(* IEC 61131-3 sources: MotionTestBenchMaster/Logical/00_AID/Libraries/Sidel_Libraries/Sidel, 28 files *)

(* ---- Types.typ ---- *)
TYPE
	AlarmCmd_Type : 	STRUCT
		ActionEn : BOOL := TRUE; (*If TRUE the action is performed; If FALSE the alarm is shown as a Message*)
		ByPassEn : BOOL;
		ByPass : BOOL;
		ActionDis : BOOL;
		Active : BOOL; (*If TRUE the alarm is activated.*)
		Visibility : BOOL := TRUE; (*If TRUE the HMI show the Alarm. The action will always performed*)
		DependentActive : BOOL; (*If TRUE the Alarm is deactivated by its master alarm V4.A.A.1.6.13*)
	END_STRUCT;
	AlarmCFG_Type : 	STRUCT
		Action : USINT;
		Category : USINT;
		OMAC_Code : UINT;
		OMAC_Index : UINT;
	END_STRUCT;
	ActionSum_Type : 	STRUCT
		Bit : UDINT;
	END_STRUCT;
	ActionSum_Enum :
		( (*V4.A.A.1.6.13*)
		ALR_NULL := 0, (*No Action, No Code*)
		ALR_MS_QuickStop := 1, (*Machine Stop: Fast deceleration ramp*)
		ALR_MS_NormalStop := 2, (*Machine Stop: Low deceleration ramp*)
		ALR_MS_QuickWithJog := 3, (*Machine Stop: Fast deceleration ramp + JOG Running Possible*)
		ALR_MS_NormalWithJog := 4, (*Machine Stop: Low deceleration ramp + JOG Running Possible*)
		ALR_MS_NormalWithJogMnt := 5, (*Machine Stop Auto Reset: Low deceleration ramp + JOG Running Possible*)
		ALR_CSR := 6, (*Container Stop Operator Reset: Immediate*)
		ALR_CSR_AfterSlowdown := 7, (*Container Stop Operator Reset: After Slowing*)
		ALR_CSR_StopAfterEmptying := 8, (*Container Stop Operator Reset: Emptying + Machine Normal Stop*)
		ALR_CSA := 9, (*Container Stop Auto Reset: Immediate*)
		ALR_CSA_AfterSlowdown := 10, (*Container Stop Auto Reset: After Slowing*)
		ALR_StartModeDisabled := 30, (*Start-Up Function Mode Disabled*)
		ALR_NoProduction := 31 (*No Action, Production Suspended (only Data Acquisition Code)*)
		);
	RCP_Management_Type : 	STRUCT
		Enable : BOOL; (*To HMI - Enable to download a recipe*)
		Started : BOOL; (*From HMI - Download Started*)
		Ended : BOOL; (*From HMI - Download Ended*)
		Received : BOOL; (*To HMI - Ended Received *)
		EditOnlineEnable : BOOL; (*To HMI - Edit Online Enabled*)
		EditOnlineActive : BOOL; (*From HMI - Edit Online Active*)
		ActiveRecipeName : STRING[70]; (*From HMI - Name of Actived Recipe*)
		RequestedRecipeName : STRING[70]; (*To HMI - Name of the requested recipe*)
		DownloadRequest : BOOL; (*To HMI - Request command to download a recipe*)
	END_STRUCT;
	RCP_Management_Step :
		(
		Wait_Download := 0,
		Download_Request := 1,
		Copy_To_Internal := 2,
		Download_Done := 3,
		Clear_Cmd := 4,
		Edit_Online := 10,
		Download_Error := 20
		);
	HMI_ITC_Page_Type : 	STRUCT
		PartnerID : USINT := 11;
		PageNum : USINT := 0;
	END_STRUCT;
	HMI_ITC_Data_Type : 	STRUCT
		PartnerID : USINT;
		ComType : USINT;
		ComAddress : STRING[35];
		ComSwap : BOOL;
		PageUp : HMI_ITC_PB_Type := (Visibility:=TRUE);
		PageDown : HMI_ITC_PB_Type := (Visibility:=TRUE);
		ComStatus : USINT;
		ComMask : HMI_ITC_SS2P_Type := (Visibility:=TRUE);
		DigitalIn : ARRAY[1..16]OF HMI_DigitalITC_Type;
		AnalogIn : ARRAY[1..4]OF HMI_AnalogITC_Type;
		DigitalOut : ARRAY[1..16]OF HMI_DigitalITC_Type;
		AnalogOut : ARRAY[1..4]OF HMI_AnalogITC_Type;
		ManActive : BOOL;
	END_STRUCT;
	HMI_AnalogITC_Type : 	STRUCT
		Visibility : BOOL;
		PV : REAL;
		Unit : STRING[10];
		Wait : BOOL;
		MinValue : REAL;
		MaxValue : REAL;
		Enable : BOOL;
		Man : BOOL;
		PV_Man : REAL;
		Description : STRING[100];
		Decimal : USINT;
	END_STRUCT;
	HMI_DigitalITC_Type : 	STRUCT
		Visibility : BOOL;
		Enable : BOOL;
		Auto : BOOL := TRUE;
		LampState : BOOL;
		Alarm : BOOL;
		Wait : BOOL;
		Man : BOOL;
		Description : STRING[100];
	END_STRUCT;
	HMI_ITC_PB_Type : 	STRUCT  (*Push button (ON-OFF;) 0=OFF - 1=ON*)
		Enable : BOOL; (*State: Command Enabled*)
		LampON : BOOL; (*State: Lamp Command ON*)
		Blink : BOOL; (*State: Blink LampOn*)
		Visibility : BOOL; (*Configuration: Present*)
		ON : BOOL; (*Command: Push Button ON*)
	END_STRUCT;
	HMI_ITC_SS2P_Type : 	STRUCT  (*Selector 2 position (Auto-Man; ON-OFF;) 0=Auto/OFF - 1=Man/ON*)
		Enable : BOOL; (*State: Command Enabled*)
		LampON : BOOL; (*State: Lamp Command ON*)
		Blink : BOOL; (*State: Blink LampOn*)
		Visibility : BOOL; (*Configuration: Present*)
		ON : BOOL; (*Command: Push Button ON*)
	END_STRUCT;
	IO_TimeClock_Type : 	STRUCT
		Seconds : UDINT;
		Nanoseconds : UDINT;
	END_STRUCT;
	Counters_Type : 	STRUCT
		CounterValue : UDINT;
		CounterTime : CounterTime_Type;
		StartDate : DINT;
	END_STRUCT;
	CounterTime_Type : 	STRUCT
		Day : UINT;
		Hour : USINT;
		Min : USINT;
		Sec : USINT;
	END_STRUCT;
	HMI_ComboBoxElements_Type : 	STRUCT
		Present : BOOL;
		Name : STRING[20];
	END_STRUCT;
	SEQ_StepConfig_Type : 	STRUCT
		T_TimePr : UINT;
		TO_TimePr : UINT;
		HMI_ID : UINT;
		TON_TimePr : UINT;
		Laps_Request : UINT;
		Cycle_Pr : UINT;
		TON_TimeSTART : BOOL;
		T_TimeSTART : BOOL;
		T_TimeSTOP : BOOL;
		T_TimeRESET : BOOL;
		Laps_Counter_Enable : BOOL;
		Cycle_RESET : BOOL;
	END_STRUCT;
	SIKO_MASTER_Type : 	STRUCT  (* *) (* *) (*13*)
		InPosition : BOOL; (*1 - The motor is in position*) (* *) (*14*)
		PositioningInProgress : BOOL; (*1 - The positioning task is in progress*) (* *) (*15*)
		CalibrationDone : BOOL; (*1 - The calibration operation is done*) (* *) (*16*)
		MotorDisabled : BOOL; (*1 - The motor is disabled*) (* *) (*17*)
		AbortPositioning : BOOL; (*1 - The current positioning is aborted*) (* *) (*18*)
		CalibrationInProgress : BOOL; (*1 - The calibration Process is in progress*) (* *) (*19*)
		Spare_06 : BOOL; (* *) (* *) (*20*)
		Spare_07 : BOOL; (* *) (* *) (*21*)
		JogForward : BOOL; (*1 - Jog Forward Command*) (* *) (*22*)
		JogBackward : BOOL; (*1 - Jog Backward Command*) (* *) (*23*)
		StartPositioning : BOOL; (*Positive Edge - Start positioning*) (* *) (*24*)
		StartRead : BOOL; (*Positive Edge - Start read parameter from the drive*) (* *) (*25*)
		StartWrite : BOOL; (*Positive Edge - Start write parameter from the drive*) (* *) (*26*)
		Calibrate : BOOL; (*Positive Edge - Calibrate command. (Calibrate value => Current pos)*) (* *) (*27*)
		Enable : BOOL; (*0 - Disable the motor; 1 - Enable motor*) (* *) (*28*)
		Spare_17 : BOOL; (* *) (* *) (*29*)
		ReadOrWriteError : BOOL; (*1 - A read or wirte error has occured*) (* *) (*30*)
		IllegalOperation : BOOL; (*1 - An illegal operation has occurred*) (* *) (*31*)
		DeviceOutsideSwLimit : BOOL; (*1 - The device is outside the sw limit*) (* *) (*32*)
		OnError : BOOL; (*1 - The motor is on error (current, temperature too high, ...)*) (* *) (*33*)
		TargetOutsideSwLimit : BOOL; (*1 - The target position is outside the sw limit (no movement is possible)*) (* *) (*34*)
		CommunicationFault : BOOL; (*1 - Comunication fault*) (* *) (*35*)
		Spare_26 : BOOL; (* *) (* *) (*36*)
		Warning : BOOL; (*1 - Warning present*) (* *) (*37*)
		EmergencyOkFbk : BOOL; (*Emergency ok feedback*) (* *) (*38*)
		WriteEnabled : BOOL; (*1 - Write process is enabled*) (* *) (*39*)
		ReadOrWriteInProgress : BOOL; (* *) (* *) (*40*)
		Spare_33 : BOOL; (* *) (* *) (*41*)
		Spare_34 : BOOL; (* *) (* *) (*42*)
		Spare_35 : BOOL; (* *) (* *) (*43*)
		Spare_36 : BOOL; (* *) (* *) (*44*)
		Spare_37 : BOOL; (* *) (* *) (*45*)
		TargetPos : REAL; (* *) (* *) (*46*)
		CurrentPos : REAL; (* *) (* *) (*47*)
		Data : SIKO_DATA_Type; (* *) (* *) (*48*)
	END_STRUCT;
	SIKO_DATA_Type : 	STRUCT  (* *) (* *) (*50*)
		OperationMode : INT; (*r/w - address:396hex - value: 2 - Don't change!!!!!!!!!!!!!!!!!!!!!!!!!!!!!!*) (* *) (*51*)
		PGain : INT; (*r/w - address:3e8hex*) (* *) (*52*)
		IGain : INT; (*r/w - address:3e9hex*) (* *) (*53*)
		DGain : INT; (*r/w - address:3eahex*) (* *) (*54*)
		VPos : INT; (*r/w - address:3echex*) (* *) (*55*)
		APos : INT; (*r/w - address:3ebhex*) (* *) (*56*)
		VJog : INT; (*r/w - address:3f0hex*) (* *) (*57*)
		SpareInt : INT; (* *) (* *) (*58*)
		GearIn : INT; (*r/w - address:3f2hex*) (* *) (*59*)
		GearOut : INT; (*r/w - address:3f3hex*) (* *) (*60*)
		SpindlePitch : INT; (*r/w - address:3f4hex*) (* *) (*61*)
		SenseOfRotation : INT; (*r/w - address:3f5hex*) (* *) (*62*)
		UpperLimit : REAL; (*r/w - address:3f8hex*) (* *) (*63*)
		LowerLimit : REAL; (*r/w - address:3f9hex*) (* *) (*64*)
		CalibrationValue : REAL; (*r/w - address:3fahex*) (* *) (*65*)
		SystemStatusWord : INT; (*r - address:3fchex*) (* *) (*66*)
		FaultBuffer0 : UINT; (*r - address:3b1 sub: 0*) (* *) (*67*)
		FaultBuffer1 : UINT; (*r - address:3b1 sub: 1*) (* *) (*68*)
		FaultBuffer2 : UINT; (*r - address:3b1 sub: 2*) (* *) (*69*)
		FaultBuffer3 : UINT; (*r - address:3b1 sub: 3*) (* *) (*70*)
		FaultBuffer4 : UINT; (*r - address:3b1 sub: 4*) (* *) (*71*)
		FaultBuffer5 : UINT; (*r - address:3b1 sub: 5*) (* *) (*72*)
		FaultBuffer6 : UINT; (*r - address:3b1 sub: 6*) (* *) (*73*)
		FaultBuffer7 : UINT; (*r - address:3b1 sub: 7*) (* *) (*74*)
		FaultBuffer8 : UINT; (*r - address:3b1 sub: 8*) (* *) (*75*)
		FaultBuffer9 : UINT; (*r - address:3b1 sub: 9*) (* *) (*76*)
		TimeoutPositioning : TIME; (* *) (* *) (*77*)
		PosWindows : REAL; (*r/w - address:3f1hex*) (* *) (*78*)
	END_STRUCT;
	SIKO_COM_Type : 	STRUCT  (* *) (* *) (*80*)
		FLR_SIKO : FLR_SIKO_Type; (* *) (* *) (*81*)
		SIKO_FLR : SIKO_FLR_Type; (* *) (* *) (*82*)
	END_STRUCT;
	FLR_SIKO_Type : 	STRUCT  (* *) (* *) (*84*)
		PKE : UINT; (* *) (* *) (*85*)
		IND : UINT; (* *) (* *) (*86*)
		PWE_H : UINT; (* *) (* *) (*87*)
		PWE_L : UINT; (* *) (* *) (*88*)
		STW : UINT; (* *) (* *) (*89*)
		HSW_H : UINT; (* *) (* *) (*90*)
		HSW_L : UINT; (* *) (* *) (*91*)
	END_STRUCT;
	SIKO_FLR_Type : 	STRUCT  (* *) (* *) (*93*)
		PKE : UINT; (* *) (* *) (*94*)
		IND : UINT; (* *) (* *) (*95*)
		PWE_H : UINT; (* *) (* *) (*96*)
		PWE_L : UINT; (* *) (* *) (*97*)
		ZSW : UINT; (* *) (* *) (*98*)
		HIW_H : UINT; (* *) (* *) (*99*)
		HIW_L : UINT; (* *) (* *) (*100*)
	END_STRUCT;
	AlarmAreaCfg_Type : 	STRUCT  (*V4.A.A.1.6.13*)
		From : UINT;
		To : UINT;
	END_STRUCT;
END_TYPE

(* ---- ComboBox.st ---- *)
FUNCTION ComboBoxString
	OUT_ComboString := '';
	FOR VAR_ElementsIndex := 0 TO 16 DO
		IF IN_ElementsStructure[VAR_ElementsIndex].Present THEN
			itoa(USINT_TO_DINT(VAR_ElementsIndex), ADR(VAR_StrIndex));
			VAR_StrComma 		:= ',';
			VAR_StrSemicolun 	:= ';';
			strcat(ADR(OUT_ComboString), ADR(VAR_StrIndex));
			strcat(ADR(OUT_ComboString), ADR(VAR_StrComma));
			strcat(ADR(OUT_ComboString), ADR(IN_ElementsStructure[VAR_ElementsIndex].Name));
			strcat(ADR(OUT_ComboString), ADR(VAR_StrSemicolun));
		END_IF
	END_FOR
	ComboBoxString := TRUE;
END_FUNCTION

(* ---- FC_Counter.st ---- *)
FUNCTION FC_Counter
	IF(IN_Clock1Hz) AND IN_TimeCondition THEN
		FC_Counter	:= TRUE;
		IN_OUT_CounterPartialStruct.CounterTime.Sec	:= IN_OUT_CounterPartialStruct.CounterTime.Sec + 1;
		IF (IN_OUT_CounterPartialStruct.CounterTime.Sec >= 60) THEN
			IN_OUT_CounterPartialStruct.CounterTime.Sec	:= 0;
			IN_OUT_CounterPartialStruct.CounterTime.Min	:= IN_OUT_CounterPartialStruct.CounterTime.Min + 1;
			IF IN_OUT_CounterPartialStruct.CounterTime.Min >= 60 THEN
				IN_OUT_CounterPartialStruct.CounterTime.Min	:= 0;
				IN_OUT_CounterPartialStruct.CounterTime.Hour	:= IN_OUT_CounterPartialStruct.CounterTime.Hour + 1;
				IF IN_OUT_CounterPartialStruct.CounterTime.Hour >= 24 THEN
					IN_OUT_CounterPartialStruct.CounterTime.Hour	:= 0;
					IN_OUT_CounterPartialStruct.CounterTime.Day	:= IN_OUT_CounterPartialStruct.CounterTime.Day + 1;
				END_IF
			END_IF
		END_IF

		IN_OUT_CounterTotalStruct.CounterTime.Sec	:= IN_OUT_CounterTotalStruct.CounterTime.Sec + 1;
		IF (IN_OUT_CounterTotalStruct.CounterTime.Sec >= 60) THEN
			IN_OUT_CounterTotalStruct.CounterTime.Sec	:= 0;
			IN_OUT_CounterTotalStruct.CounterTime.Min	:= IN_OUT_CounterTotalStruct.CounterTime.Min + 1;
			IF IN_OUT_CounterTotalStruct.CounterTime.Min >= 60 THEN
				IN_OUT_CounterTotalStruct.CounterTime.Min	:= 0;
				IN_OUT_CounterTotalStruct.CounterTime.Hour	:= IN_OUT_CounterTotalStruct.CounterTime.Hour + 1;
				IF IN_OUT_CounterTotalStruct.CounterTime.Hour >= 24 THEN
					IN_OUT_CounterTotalStruct.CounterTime.Hour	:= 0;
					IN_OUT_CounterTotalStruct.CounterTime.Day	:= IN_OUT_CounterTotalStruct.CounterTime.Day + 1;
				END_IF
			END_IF
		END_IF
	END_IF

	IF IN_IncrementCondition THEN
		FC_Counter	:= TRUE;
		IN_OUT_CounterPartialStruct.CounterValue	:= IN_OUT_CounterPartialStruct.CounterValue + 1;
		IN_OUT_CounterTotalStruct.CounterValue		:= IN_OUT_CounterTotalStruct.CounterValue + 1;
	END_IF

	IF IN_Reset THEN
		FC_Counter	:= TRUE;
		IN_OUT_CounterPartialStruct.CounterTime.Sec		:= 0;
		IN_OUT_CounterPartialStruct.CounterTime.Min		:= 0;
		IN_OUT_CounterPartialStruct.CounterTime.Hour	:= 0;
		IN_OUT_CounterPartialStruct.CounterTime.Day		:= 0;
		IN_OUT_CounterPartialStruct.CounterValue		:= 0;
		IN_OUT_CounterPartialStruct.StartDate			:= DT_TO_DINT(IN_Date);
	ELSIF IN_OUT_CounterPartialStruct.StartDate = 0 THEN
		IN_OUT_CounterPartialStruct.StartDate		:= DT_TO_DINT(IN_Date);
	ELSIF IN_OUT_CounterTotalStruct.StartDate	= 0 THEN
		IN_OUT_CounterTotalStruct.StartDate		:= DT_TO_DINT(IN_Date);
	END_IF
END_FUNCTION

(* ---- FC_Parity.st ---- *)
FUNCTION FC_Parity
	FC_Parity := NOT IN_Value.0;
END_FUNCTION

(* ---- FC_Reminder.st ---- *)
(* Reminder With Minimum Value *)
FUNCTION FC_ReminderShift
	LocalDivisor	:= SEL(Divisor<>0, 1, Divisor);

	ReminderA	:= (Dividend - ((Dividend / LocalDivisor) * LocalDivisor));
	ReminderB	:= (ReminderA + Divisor - ((ReminderA + LocalDivisor) / LocalDivisor) * LocalDivisor);
	ReminderC	:= (ReminderB + Start - ((ReminderB + Start) / LocalDivisor) * LocalDivisor);

	FC_ReminderShift	:= SEL(ReminderC <> 0, LocalDivisor, ReminderC);
END_FUNCTION

(* ---- FC_SpeedCheck.st ---- *)
FUNCTION FC_SpeedCheck
	CASE IN_Mode OF
		CST_EQ:	(* Actual speed equal to requested *)
			FC_SpeedCheck := (IN_SpeedAct >= (IN_SpeedReq * 0.9)) AND (IN_SpeedAct <= (IN_SpeedReq / 0.9));

		CST_GE:	(* Actual speed greater then requested *)
			FC_SpeedCheck := IN_SpeedAct >= IN_SpeedReq * 0.9;

		CST_LE:	(* Actual speed lower then requested *)
			FC_SpeedCheck := IN_SpeedAct <= IN_SpeedReq / 0.9;

		CST_GT:	(* Actual speed greater then requested *)
			FC_SpeedCheck := IN_SpeedAct > IN_SpeedReq * 0.9;

		CST_LT:	(* Actual speed lower then requested *)
			FC_SpeedCheck := IN_SpeedAct < IN_SpeedReq / 0.9;

		ELSE
			FC_SpeedCheck := FALSE;
	END_CASE
END_FUNCTION

(* ---- FC_Timer.st ---- *)
FUNCTION FC_IncTimer
	IF IN_Reset THEN
		FC_IncTimer	:= TRUE;
		IN_OUT_CounterStruct.Sec	:= 0;
		IN_OUT_CounterStruct.Min	:= 0;
		IN_OUT_CounterStruct.Hour	:= 0;
		IN_OUT_CounterStruct.Day	:= 0;
	ELSIF(IN_Clock1Hz) AND IN_Condition THEN
		FC_IncTimer	:=	TRUE;
		IN_OUT_CounterStruct.Sec	:= IN_OUT_CounterStruct.Sec + 1;
		IF (IN_OUT_CounterStruct.Sec >= 60) THEN
			IN_OUT_CounterStruct.Sec	:= 0;
			IN_OUT_CounterStruct.Min	:= IN_OUT_CounterStruct.Min + 1;
			IF IN_OUT_CounterStruct.Min >= 60 THEN
				IN_OUT_CounterStruct.Min	:= 0;
				IN_OUT_CounterStruct.Hour	:= IN_OUT_CounterStruct.Hour + 1;
				IF IN_OUT_CounterStruct.Hour >= 24 THEN
					IN_OUT_CounterStruct.Hour	:= 0;
					IN_OUT_CounterStruct.Day	:= IN_OUT_CounterStruct.Day + 1;
				END_IF
			END_IF
		END_IF
	ELSE
		FC_IncTimer	:= FALSE;
	END_IF
END_FUNCTION

FUNCTION FC_MacaoTimer
	IF IN_Reset THEN
		IN_OUT_Counter	:= 0;
	ELSIF IN_Clock1Hz AND IN_Condition THEN
		IN_OUT_Counter	:= IN_OUT_Counter + 1;
	END_IF
	FC_MacaoTimer := TRUE;
END_FUNCTION

(* ---- LftConAirPress.st ---- *)
FUNCTION LftConAirPressSp
	VAR_PistonSurface 	:= amPI * (EXPT(CST_PistonDiameterExt, 2) - EXPT(CST_PistonDiameterInt, 2)) / 4.0;
	VAR_DeltaPProduct 	:= (EXPT(57.0, 2) - EXPT(RcpCanDiameter, 2)) * amPI / 4.0 * RcpPressureSp / 10.0;
	VAR_DeltaPrexPist  	:= (ABS(VAR_DeltaPProduct * 1000000.0 / VAR_PistonSurface / 100000.0)) * BOOL_TO_REAL((RcpCanDiameter > 57.0));
	VAR_PbasePiston 	:= CST_PistonSpringStrengthRse / (VAR_PistonSurface / 100.0) / 10;
	LftConAirPressSp	:= VAR_PbasePiston + VAR_DeltaPrexPist + 1.5;
END_FUNCTION

(* ---- AlarmScheduler.st ---- *)
FUNCTION_BLOCK AlarmScheduler
	//V4.A.A.1.6.13
	memset(ADR(AlarmActionTemp), 0, SIZEOF(AlarmActionTemp));

	FOR x := 0 TO 24 DO//V1.7.2
		IF AlarmAreaCfg[x].From = 0 OR AlarmAreaCfg[x].To = 0 THEN
		ELSE
			FOR i := MAX(0, AlarmAreaCfg[x].From - 1) TO MAX(AlarmAreaCfg[x].To - 1, AlarmAreaCfg[x].From - 1) DO

				Alarm ACCESS AdrAlarm + (SIZEOF(Alarm) * i);
				AlarmCFG ACCESS AdrAlarmCFG + (SIZEOF(AlarmCFG) * i);
				AlarmOldStatus ACCESS AdrAlarmOldStatus + (SIZEOF(AlarmOldStatus) * i);
				HMI ACCESS AdrHMI + (SIZEOF(HMI) * i);

				IF FirstAlarmActive.OMAC_Index = AlarmCFG.OMAC_Index THEN
					memset(ADR(FirstAlarmActive), 0, SIZEOF(FirstAlarmActive));
				END_IF

				IF FirstExternalAlarmActive.OMAC_Index = AlarmCFG.OMAC_Index THEN
					memset(ADR(FirstExternalAlarmActive), 0, SIZEOF(FirstExternalAlarmActive));
				END_IF

				IF FirstAlarmActive.OMAC_Index = 0      AND Alarm.Active AND
					(Alarm.ActionEn AND NOT Alarm.ByPass) AND
					(AlarmCFG.Action <> 0) AND (AlarmCFG.Action <> 67) AND
					NOT Alarm.DependentActive THEN
					FirstAlarmActive := AlarmCFG;
				END_IF

				IF FirstExternalAlarmActive.OMAC_Index = 0      AND Alarm.Active AND
					(Alarm.ActionEn AND NOT Alarm.ByPass) AND
					(AlarmCFG.Action <> 0) AND (AlarmCFG.Category = 3) AND
					NOT Alarm.DependentActive THEN
					FirstExternalAlarmActive := AlarmCFG;
				END_IF

				IF Alarm.Active AND (Alarm.ActionEn AND NOT Alarm.ByPass AND Alarm.Visibility) AND
					NOT AlarmOldStatus AND NOT CriticalAcknoledgeRequest AND
					(AlarmCFG.Action > 0 AND AlarmCFG.Action < 32)	AND
					NOT Alarm.DependentActive THEN
					CriticalAcknoledgeRequest := AlarmCFG.Action <> 6; //ALARM SCHEDULER V4_03:ESCLUSIONE DEGLI ALLARMI DI SBLOCCO PORTE
				END_IF

				IF Alarm.Active AND (Alarm.ActionEn AND NOT Alarm.ByPass AND Alarm.Visibility) AND
					NOT AlarmOldStatus AND NOT AlarmAcknoledgeRequest AND
					(AlarmCFG.Action >= 32 AND AlarmCFG.Action < 64)	AND
					NOT Alarm.DependentActive THEN
					AlarmAcknoledgeRequest := TRUE;
				END_IF

				Alarm.ActionDis := NOT Alarm.ActionEn;

				HMI.0			:= Alarm.ActionEn;
				HMI.1			:= Alarm.ByPassEn;
				HMI.2;
				HMI.3;
				Alarm.ByPass	:= HMI.4;
				HMI.5			:= Alarm.ActionDis;
				HMI.6			:= Alarm.Active;
				HMI.7			:= Alarm.Visibility;

				CASE AlarmCFG.Action OF

					0:
						AlarmActionTemp.Bit.ALR_NULL					:= Alarm.Active AND NOT Alarm.DependentActive OR AlarmActionTemp.Bit.ALR_NULL;
					1:
						AlarmActionTemp.Bit.ALR_MS_QuickStop			:= Alarm.Active AND (Alarm.ActionEn AND NOT Alarm.ByPass AND NOT Alarm.DependentActive) OR AlarmActionTemp.Bit.ALR_MS_QuickStop;
					2:
						AlarmActionTemp.Bit.ALR_MS_NormalStop			:= Alarm.Active AND (Alarm.ActionEn AND NOT Alarm.ByPass AND NOT Alarm.DependentActive) OR AlarmActionTemp.Bit.ALR_MS_NormalStop;
					3:
						AlarmActionTemp.Bit.ALR_MS_QuickWithJog			:= Alarm.Active AND (Alarm.ActionEn AND NOT Alarm.ByPass AND NOT Alarm.DependentActive) OR AlarmActionTemp.Bit.ALR_MS_QuickWithJog;
					4:
						AlarmActionTemp.Bit.ALR_MS_NormalWithJog		:= Alarm.Active AND (Alarm.ActionEn AND NOT Alarm.ByPass AND NOT Alarm.DependentActive) OR AlarmActionTemp.Bit.ALR_MS_NormalWithJog;
					6:
						AlarmActionTemp.Bit.ALR_MS_NormalWithJogMnt		:= Alarm.Active AND (Alarm.ActionEn AND NOT Alarm.ByPass AND NOT Alarm.DependentActive) OR AlarmActionTemp.Bit.ALR_MS_NormalWithJogMnt;
					10:
						AlarmActionTemp.Bit.ALR_CSR_StopAfterEmptying	:= Alarm.Active AND (Alarm.ActionEn AND NOT Alarm.ByPass AND NOT Alarm.DependentActive) OR AlarmActionTemp.Bit.ALR_CSR_StopAfterEmptying;
					32:
						AlarmActionTemp.Bit.ALR_CSR						:= Alarm.Active AND (Alarm.ActionEn AND NOT Alarm.ByPass AND NOT Alarm.DependentActive) OR AlarmActionTemp.Bit.ALR_CSR;
					33:
						AlarmActionTemp.Bit.ALR_CSR_AfterSlowdown		:= Alarm.Active AND (Alarm.ActionEn AND NOT Alarm.ByPass AND NOT Alarm.DependentActive) OR AlarmActionTemp.Bit.ALR_CSR_AfterSlowdown;
					64:
						AlarmActionTemp.Bit.ALR_CSA						:= Alarm.Active AND (Alarm.ActionEn AND NOT Alarm.ByPass AND NOT Alarm.DependentActive) OR AlarmActionTemp.Bit.ALR_CSA;
					65:
						AlarmActionTemp.Bit.ALR_CSA_AfterSlowdown		:= Alarm.Active AND (Alarm.ActionEn AND NOT Alarm.ByPass AND NOT Alarm.DependentActive) OR AlarmActionTemp.Bit.ALR_CSA_AfterSlowdown;
					81:
						AlarmActionTemp.Bit.ALR_StartModeDisabled		:= Alarm.Active AND (Alarm.ActionEn AND NOT Alarm.ByPass AND NOT Alarm.DependentActive) OR AlarmActionTemp.Bit.ALR_StartModeDisabled;
					86:
						AlarmActionTemp.Bit.ALR_NoProduction			:= Alarm.Active AND (Alarm.ActionEn AND NOT Alarm.ByPass AND NOT Alarm.DependentActive) OR AlarmActionTemp.Bit.ALR_NoProduction;

					ELSE
						AlarmActionTemp.Bit.ALR_NULL					:= Alarm.Active AND NOT Alarm.DependentActive OR AlarmActionTemp.Bit.ALR_NULL;
				END_CASE

				//EXTRACTION OF FIRST ALARM FOR EACH CATEGORY
				IF FirstCriticalAlarmActive.OMAC_Index = AlarmCFG.OMAC_Index THEN//V4.A.A.1.7.0
					memset(ADR(FirstCriticalAlarmActive), 0, SIZEOF(FirstCriticalAlarmActive));
				END_IF

				IF FirstAlertAlarmActive.OMAC_Index = AlarmCFG.OMAC_Index THEN//V4.A.A.1.7.0
					memset(ADR(FirstAlertAlarmActive), 0, SIZEOF(FirstAlertAlarmActive));
				END_IF

				IF FirstExtCriticalAlarmActive.OMAC_Index = AlarmCFG.OMAC_Index THEN//V4.A.A.1.7.0
					memset(ADR(FirstExtCriticalAlarmActive), 0, SIZEOF(FirstExtCriticalAlarmActive));
				END_IF

				IF FirstExtAlertAlarmActive.OMAC_Index = AlarmCFG.OMAC_Index THEN//V4.A.A.1.7.0
					memset(ADR(FirstExtAlertAlarmActive), 0, SIZEOF(FirstExtAlertAlarmActive));
				END_IF
				IF FirstCsAlarmActive.OMAC_Index = AlarmCFG.OMAC_Index THEN//V4.A.A.1.7.0
					memset(ADR(FirstCsAlarmActive), 0, SIZEOF(FirstCsAlarmActive));
				END_IF
				//V4.A.A.1.7.0
				IF FirstCriticalAlarmActive.OMAC_Index = 0	AND Alarm.Active		AND
					(Alarm.ActionEn					AND NOT Alarm.ByPass)		AND
					(AlarmCFG.Action > 0)			AND (AlarmCFG.Action <= 31)	AND (AlarmCFG.Category <> 3) AND
					NOT Alarm.DependentActive THEN
					FirstCriticalAlarmActive := AlarmCFG;
				END_IF
				//V4.A.A.1.7.0
				IF FirstAlertAlarmActive.OMAC_Index = 0	AND Alarm.Active			AND
					(Alarm.ActionEn					AND NOT Alarm.ByPass)		AND
					(AlarmCFG.Action >= 32)			AND (AlarmCFG.Action <= 63)	AND (AlarmCFG.Category <> 3) AND
					NOT Alarm.DependentActive THEN
					FirstAlertAlarmActive := AlarmCFG;
				END_IF
				//V4.A.A.1.7.0
				IF FirstExtCriticalAlarmActive.OMAC_Index = 0	AND Alarm.Active			AND
					(Alarm.ActionEn							AND NOT Alarm.ByPass)		AND
					(AlarmCFG.Action > 0)			AND (AlarmCFG.Action <= 31)	AND (AlarmCFG.Category = 3)	AND
					NOT Alarm.DependentActive THEN
					FirstExtCriticalAlarmActive := AlarmCFG;
				END_IF
				//V4.A.A.1.7.0
				IF FirstExtAlertAlarmActive.OMAC_Index = 0	AND Alarm.Active			AND
					(Alarm.ActionEn							AND NOT Alarm.ByPass)		AND
					(AlarmCFG.Action >= 32)			AND (AlarmCFG.Action <= 63)	AND (AlarmCFG.Category = 3)	AND
					NOT Alarm.DependentActive THEN
					FirstExtAlertAlarmActive := AlarmCFG;
				END_IF
				//V4.A.A.1.7.0
				IF FirstCsAlarmActive.OMAC_Index = 0	AND Alarm.Active			AND
					(Alarm.ActionEn							AND NOT Alarm.ByPass)		AND
					(AlarmCFG.Action >= 64)			AND (AlarmCFG.Action <= 65)	AND
					NOT Alarm.DependentActive THEN
					FirstCsAlarmActive := AlarmCFG;
				END_IF
				//END EXTRACTION

				AlarmOldStatus := Alarm.Active AND (Alarm.ActionEn AND NOT Alarm.ByPass AND NOT Alarm.DependentActive);
			END_FOR
		END_IF
	END_FOR

	AlarmAction	:= AlarmActionTemp;
END_FUNCTION_BLOCK

FUNCTION_BLOCK FirstAlarmCombiner
	IF (FirstAlarmActive.OMAC_Index >= SkidAlarmFrom) AND (FirstAlarmActive.OMAC_Index <= SkidAlarmTo) THEN
		memset(ADR(FirstAlarmActive), 0, SIZEOF(FirstAlarmActive));
	END_IF

	IF (FirstExternalAlarmActive.OMAC_Index >= SkidAlarmFrom) AND (FirstExternalAlarmActive.OMAC_Index <= SkidAlarmTo) THEN
		memset(ADR(FirstExternalAlarmActive), 0, SIZEOF(FirstExternalAlarmActive));
	END_IF

	IF SkidFirstAlarm <> 0 AND FirstAlarmActive.OMAC_Index = 0 THEN
		FirstAlarmActive.OMAC_Index := SkidFirstAlarm;
	END_IF

	IF SkidFirstExternalAlarm <> 0 AND FirstExternalAlarmActive.OMAC_Index = 0 THEN
		FirstExternalAlarmActive.OMAC_Index := SkidFirstExternalAlarm;
	END_IF
END_FUNCTION_BLOCK

(* ---- AnalogTotalizer.st ---- *)
FUNCTION_BLOCK AnalogTotalizer
	RTInfo(enable := TRUE);

	CASE IN_ConfigType OF
		0:
			VAR_AuxPulse := IN_PulseWeight * BOOL_TO_REAL(EDGEPOS(IN_Pulse));
		1:
			VAR_AuxPulse := IN_AnalogPV * UDINT_TO_REAL(RTInfo.cycle_time) /1000000;
		2:
			VAR_AuxPulse := IN_AnalogPV * UDINT_TO_REAL(RTInfo.cycle_time) /1000000 / 60;
		3:
			VAR_AuxPulse := IN_AnalogPV * UDINT_TO_REAL(RTInfo.cycle_time) /1000000 / 3600;
	END_CASE

	OUT_TotalCounter := VAR_AuxPulse + OUT_TotalCounter;

	IF IN_Reset THEN
		OUT_TotalCounter := 0.0;
	END_IF
END_FUNCTION_BLOCK

(* ---- Blink.st ---- *)
FUNCTION_BLOCK FB_Blinker
	VAR_TimeValue	:= REAL_TO_TIME((1.0 / IN_Freq) * 1000);

	TMR_TON_OnDelay(IN:= NOT OUT,	PT:= VAR_TimeValue / 2);
	TMR_TON_OffDelay(IN:= OUT,		PT:= VAR_TimeValue / 2);

	IF TMR_TON_OnDelay.Q THEN
		OUT	:= TRUE;
	ELSIF TMR_TON_OffDelay.Q THEN
		OUT	:= FALSE;
	END_IF
END_FUNCTION_BLOCK

(* ---- CyclicActivation.st ---- *)
FUNCTION_BLOCK CyclicActivation
	VAR_RtInfo(enable:=TRUE);
	VAR_CycleCounter	:= MAX(1, VAR_CycleCounter + 1);
	OUT_A	:= FALSE;
	OUT_B	:= FALSE;

	TMR_TON_CycleA(	IN := VAR_Cycle,
	PT := (IN_CycleTime / 2) - UDINT_TO_TIME(VAR_RtInfo.cycle_time / 1000));

	TMR_TON_CycleB(	IN := NOT VAR_Cycle,
	PT := (IN_CycleTime / 2) - UDINT_TO_TIME(VAR_RtInfo.cycle_time / 1000));

	IF TMR_TON_CycleA.Q THEN
		OUT_A		:= TRUE;
		VAR_Cycle	:= FALSE;
	ELSIF TMR_TON_CycleB.Q THEN
		OUT_B		:= TRUE;
		VAR_Cycle	:= TRUE;
	ELSE
		RETURN;
	END_IF

	VAR_CycleTime	:= (UDINT_TO_REAL(VAR_RtInfo.cycle_time) * VAR_CycleCounter) / 1000000.0;
	VAR_CycleCounter 	:= 0.0;
	memset(ADR(TMR_TON_CycleA), 0, SIZEOF(TMR_TON_CycleA));
	memset(ADR(TMR_TON_CycleB), 0, SIZEOF(TMR_TON_CycleB));
END_FUNCTION_BLOCK

(* ---- FB_Counter.st ---- *)
FUNCTION_BLOCK FB_Counter
	IF(IN_Clock1Hz) AND IN_TimeCondition THEN
		IN_OUT_CounterPartialStruct.CounterTime.Sec	:= IN_OUT_CounterPartialStruct.CounterTime.Sec + 1;
		IF (IN_OUT_CounterPartialStruct.CounterTime.Sec >= 60) THEN
			IN_OUT_CounterPartialStruct.CounterTime.Sec	:= 0;
			IN_OUT_CounterPartialStruct.CounterTime.Min	:= IN_OUT_CounterPartialStruct.CounterTime.Min + 1;
			IF IN_OUT_CounterPartialStruct.CounterTime.Min >= 60 THEN
				IN_OUT_CounterPartialStruct.CounterTime.Min	:= 0;
				IN_OUT_CounterPartialStruct.CounterTime.Hour	:= IN_OUT_CounterPartialStruct.CounterTime.Hour + 1;
				IF IN_OUT_CounterPartialStruct.CounterTime.Hour >= 24 THEN
					IN_OUT_CounterPartialStruct.CounterTime.Hour	:= 0;
					IN_OUT_CounterPartialStruct.CounterTime.Day	:= IN_OUT_CounterPartialStruct.CounterTime.Day + 1;
				END_IF
			END_IF
		END_IF

		IN_OUT_CounterTotalStruct.CounterTime.Sec	:= IN_OUT_CounterTotalStruct.CounterTime.Sec + 1;
		IF (IN_OUT_CounterTotalStruct.CounterTime.Sec >= 60) THEN
			IN_OUT_CounterTotalStruct.CounterTime.Sec	:= 0;
			IN_OUT_CounterTotalStruct.CounterTime.Min	:= IN_OUT_CounterTotalStruct.CounterTime.Min + 1;
			IF IN_OUT_CounterTotalStruct.CounterTime.Min >= 60 THEN
				IN_OUT_CounterTotalStruct.CounterTime.Min	:= 0;
				IN_OUT_CounterTotalStruct.CounterTime.Hour	:= IN_OUT_CounterTotalStruct.CounterTime.Hour + 1;
				IF IN_OUT_CounterTotalStruct.CounterTime.Hour >= 24 THEN
					IN_OUT_CounterTotalStruct.CounterTime.Hour	:= 0;
					IN_OUT_CounterTotalStruct.CounterTime.Day	:= IN_OUT_CounterTotalStruct.CounterTime.Day + 1;
				END_IF
			END_IF
		END_IF
	END_IF

	IF IN_IncrementCondition THEN
		tempReal := tempReal + IN_PulseWeight;
		IF tempReal >= 1.0 THEN
			IN_OUT_CounterPartialStruct.CounterValue	:= IN_OUT_CounterPartialStruct.CounterValue + TRUNC(tempReal);
			IN_OUT_CounterTotalStruct.CounterValue		:= IN_OUT_CounterTotalStruct.CounterValue 	+ TRUNC(tempReal);
			tempReal := tempReal - (TRUNC(tempReal));
		END_IF
	END_IF

	IF IN_Reset THEN
		IN_OUT_CounterPartialStruct.CounterTime.Sec		:= 0;
		IN_OUT_CounterPartialStruct.CounterTime.Min		:= 0;
		IN_OUT_CounterPartialStruct.CounterTime.Hour	:= 0;
		IN_OUT_CounterPartialStruct.CounterTime.Day		:= 0;
		IN_OUT_CounterPartialStruct.CounterValue		:= 0;
		IN_OUT_CounterPartialStruct.StartDate			:= DT_TO_DINT(IN_Date);
	ELSIF IN_OUT_CounterPartialStruct.StartDate = 0 THEN
		IN_OUT_CounterPartialStruct.StartDate		:= DT_TO_DINT(IN_Date);
	ELSIF IN_OUT_CounterTotalStruct.StartDate	= 0 THEN
		IN_OUT_CounterTotalStruct.StartDate		:= DT_TO_DINT(IN_Date);
	END_IF
END_FUNCTION_BLOCK

(* ---- FB_Flip.st ---- *)
FUNCTION_BLOCK FB_Flip
	TON_Blink.IN := NOT TON_Blink.Q;
	TON_Blink.PT := t#1s;
	TON_Blink();

	IF EDGEPOS(TON_Blink.Q) THEN
		VAR_CyleOn 		:= FALSE;
		VAR_CyleCntOn	:= FALSE;
		VAR_CyleCntOff	:= FALSE;
		VAR_CyleOnTimeReset := FALSE;
		VAR_CyleOffTimeReset:= FALSE;
		VAR_CyleNrReset	:= FALSE;
		VAR_CycleNrDone	:= FALSE;
		CASE Command_State OF
			0:
				IF IN_CycleOn AND NOT IN_CyclePause THEN
					IF IN_CycleStartOffCount THEN
						Command_State := 2;
					ELSIF IN_CycleTimeOn > 0 THEN
						Command_State := 1;
					END_IF
				END_IF

			1:	//ON TIME
				VAR_CyleOn 		:= TRUE;
				VAR_CyleCntOn	:= TRUE;
				VAR_CyleOffTimeReset	:= TRUE;

				IF NOT IN_CycleOn THEN
					Command_State := 99; // //RESET CNT
				ELSIF IN_CyclePause THEN
					Command_State := 10; // PAUSE CMD
				ELSE
					IF VAR_CycleOnDone THEN
						VAR_CyleOnTimeReset := TRUE;
						IF IN_CycleLoop THEN
							IF IN_CycleTimeOff > 0 THEN
								Command_State := 2; //PAUSE TIME
							END_IF
						ELSE
							VAR_CycleNr 	:= MIN(VAR_CycleNr  +1, IN_CycleNr);
							 IF (IN_CycleNr = VAR_CycleNr) AND NOT IN_CycleLoop THEN
								Command_State := 3; // DONE
							ELSE
								Command_State := 2; //PAUSE TIME
							END_IF
						END_IF
					END_IF
				END_IF

			2: //PAUSE TIME

				VAR_CyleCntOff	:= NOT IN_CyclePause;
				VAR_CyleOnTimeReset	:= TRUE;

				IF NOT IN_CycleOn THEN
					Command_State := 99; // //RESET CNT
				ELSIF VAR_CycleOffDone AND NOT IN_CyclePause THEN
					VAR_CyleOffTimeReset := TRUE;
					IF VAR_CycleNrDone THEN
						Command_State := 3; // DONE
					ELSIF IN_CycleTimeOn > 0 THEN
						Command_State := 1; // ON TIME
					END_IF
				END_IF

			3: // DONE
				VAR_CycleNrDone	:= TRUE;
				IF NOT IN_CycleOn OR IN_CycleLoop THEN
					Command_State := 99; // //RESET CNT
				END_IF

			10: // PAUSE

				IF NOT IN_CycleOn THEN
					Command_State := 99; // //RESET CNT
				ELSIF NOT IN_CyclePause THEN
					Command_State := 1; // OFF
				END_IF

			99: //RESET CNT
				VAR_CyleOnTimeReset := TRUE;
				VAR_CyleOffTimeReset:= TRUE;
				VAR_CycleNr := 0;
				Command_State := 0; // OFF
		END_CASE

		IF VAR_CyleCntOn THEN
			VAR_CycleTimeOn := MIN(VAR_CycleTimeOn  +1, IN_CycleTimeOn);
			VAR_CycleOnDone := IN_CycleTimeOn = VAR_CycleTimeOn;
		ELSE
			VAR_CycleOnDone := FALSE;
		END_IF

		IF VAR_CyleCntOff THEN
			VAR_CycleTimeOff := MIN(VAR_CycleTimeOff +1, IN_CycleTimeOff);
			VAR_CycleOffDone := IN_CycleTimeOff = VAR_CycleTimeOff;
		ELSE
			VAR_CycleOffDone := FALSE;
		END_IF

		IF VAR_CyleOffTimeReset THEN
			VAR_CycleTimeOff := 0;
		END_IF
		IF VAR_CyleOnTimeReset THEN
			VAR_CycleTimeOn := 0;
		END_IF
		IF IN_CycleNrReset THEN
			VAR_CycleNr 	:= 0;
		END_IF

		Out 			:= VAR_CyleOn;
		OUT_CycleNr		:= VAR_CycleNr;
		OUT_CycleTimeOn	:= VAR_CycleTimeOn;
		OUT_CycleTimeOff:= VAR_CycleTimeOff;
		OUT_CycleDone 	:= VAR_CycleNrDone;
	END_IF
END_FUNCTION_BLOCK

(* ---- FB_ITC.st ---- *)
FUNCTION_BLOCK FB_HMI_ITC_DigitalBool
	VAR_ProgressiveId := INT_TO_UINT(FC_ReminderShift(UINT_TO_INT(Index), 16, 0));

	IF IN_ReadOnly OR IN_HMIAutoForce THEN
		VAR_Auto	:= TRUE;
		VAR_Man		:= FALSE;
	END_IF

	IF IN_IOType THEN
		ITC_IO 	:= SEL(VAR_Auto, VAR_Man, ITC);
	ELSE
		ITC 	:= SEL(VAR_Auto, VAR_Man, ITC_IO);
	END_IF

	IF VAR_OldPage <> HMI_Page.PageNum THEN
		VAR_PageSwitch	:= TRUE;
	END_IF

	IF (Index = (VAR_ProgressiveId + 16 * HMI_Page.PageNum)) AND IN_Visibility THEN
		IF VAR_PageSwitch THEN
			IF IN_IOType THEN
				HMI_Data.DigitalOut[VAR_ProgressiveId].Auto	:= VAR_Auto;
				HMI_Data.DigitalOut[VAR_ProgressiveId].Man	:= VAR_Man;
			ELSE
				HMI_Data.DigitalIn[VAR_ProgressiveId].Auto	:= VAR_Auto;
				HMI_Data.DigitalIn[VAR_ProgressiveId].Man	:= VAR_Man;
			END_IF
			VAR_PageSwitch	:= FALSE;
		END_IF

		IF IN_IOType THEN
			HMI_Data.DigitalOut[VAR_ProgressiveId].Visibility	:= IN_Visibility;
			HMI_Data.DigitalOut[VAR_ProgressiveId].Enable		:= NOT IN_ReadOnly AND NOT IN_HMIAutoForce;
			HMI_Data.DigitalOut[VAR_ProgressiveId].LampState	:= ITC_IO;
			HMI_Data.DigitalOut[VAR_ProgressiveId].Wait			:= IN_Wait;
			HMI_Data.DigitalOut[VAR_ProgressiveId].Alarm		:= IN_Alarm;
			HMI_Data.DigitalOut[VAR_ProgressiveId].Description	:= IN_Description;

			IF EDGEPOS(HMI_Data.DigitalOut[VAR_ProgressiveId].Auto) THEN
				HMI_Data.DigitalOut[VAR_ProgressiveId].Man := FALSE;
			ELSIF EDGEPOS(HMI_Data.DigitalOut[VAR_ProgressiveId].Man) THEN
				HMI_Data.DigitalOut[VAR_ProgressiveId].Auto := FALSE;
			END_IF

			IF IN_ReadOnly OR IN_HMIAutoForce THEN
				HMI_Data.DigitalOut[VAR_ProgressiveId].Auto	:= TRUE;
				HMI_Data.DigitalOut[VAR_ProgressiveId].Man	:= FALSE;
			END_IF

			VAR_Auto	:= HMI_Data.DigitalOut[VAR_ProgressiveId].Auto;
			VAR_Man		:= HMI_Data.DigitalOut[VAR_ProgressiveId].Man;
		ELSE
			HMI_Data.DigitalIn[VAR_ProgressiveId].Visibility	:= IN_Visibility;
			HMI_Data.DigitalIn[VAR_ProgressiveId].Enable		:= NOT IN_ReadOnly AND NOT IN_HMIAutoForce;
			HMI_Data.DigitalIn[VAR_ProgressiveId].LampState 	:= ITC;
			HMI_Data.DigitalIn[VAR_ProgressiveId].Wait			:= IN_Wait;
			HMI_Data.DigitalIn[VAR_ProgressiveId].Alarm			:= IN_Alarm;
			HMI_Data.DigitalIn[VAR_ProgressiveId].Description	:= IN_Description;

			IF EDGEPOS(HMI_Data.DigitalIn[VAR_ProgressiveId].Auto) THEN
				HMI_Data.DigitalIn[VAR_ProgressiveId].Man := FALSE;
			ELSIF EDGEPOS(HMI_Data.DigitalIn[VAR_ProgressiveId].Man) THEN
				HMI_Data.DigitalIn[VAR_ProgressiveId].Auto := FALSE;
			END_IF

			IF IN_ReadOnly OR IN_HMIAutoForce THEN
				HMI_Data.DigitalIn[VAR_ProgressiveId].Auto	:= TRUE;
				HMI_Data.DigitalIn[VAR_ProgressiveId].Man	:= FALSE;
			END_IF

			VAR_Auto	:= HMI_Data.DigitalIn[VAR_ProgressiveId].Auto;
			VAR_Man		:= HMI_Data.DigitalIn[VAR_ProgressiveId].Man;
		END_IF
	ELSIF (Index < (VAR_ProgressiveId + 16 * HMI_Page.PageNum)) THEN
		IF IN_IOType THEN
			HMI_Data.DigitalOut[VAR_ProgressiveId].Visibility	:= FALSE;
		ELSE
			HMI_Data.DigitalIn[VAR_ProgressiveId].Visibility	:= FALSE;
		END_IF
	END_IF

	VAR_OldPage := HMI_Page.PageNum;

	HMI_Data.ManActive	:= NOT VAR_Auto OR HMI_Data.ManActive;

	IF (Index > (16 + 16 * HMI_Page.PageNum)) AND IN_Visibility THEN
		HMI_Data.PageUp.Enable := TRUE;
	END_IF

	IF HMI_Page.PageNum <> 0 THEN
		HMI_Data.PageDown.Enable := TRUE;
	END_IF

	OUT_Man			:= NOT VAR_Auto;
	OUT_ManValue	:= VAR_Man;
	Index			:= Index + 1;
END_FUNCTION_BLOCK

FUNCTION_BLOCK FB_HMI_ITC_DigitalByte
	VAR_ProgressiveId := INT_TO_UINT(FC_ReminderShift(UINT_TO_INT(Index), 16, 0));

	IF IN_ReadOnly OR IN_HMIAutoForce THEN
		VAR_Auto	:= TRUE;
		VAR_Man		:= FALSE;
	END_IF

	IF IN_IOType THEN
		FOR VAR_BitIndex := 0 TO 7 DO
			IF VAR_BitIndex = INT_TO_USINT(IN_BitNumber) THEN
				IF NOT VAR_Auto THEN
					VAR_BitArray[VAR_BitIndex] := VAR_Man;
				ELSE
					VAR_BitArray[VAR_BitIndex] := ITC;
				END_IF
			ELSE
				VAR_BitArray[VAR_BitIndex] := (ITC_IO AND REAL_TO_BYTE(pow(2, VAR_BitIndex))) <> 0;
			END_IF
		END_FOR

		ITC_IO	:= 0;

		FOR VAR_BitIndex := 0 TO 7 DO
			ITC_IO	:= ITC_IO OR UINT_TO_BYTE(((REAL_TO_UINT(pow(2, VAR_BitIndex))) * VAR_BitArray[VAR_BitIndex]));
		END_FOR
	ELSE
		IF NOT VAR_Auto THEN
			ITC		:= VAR_Man;
		ELSE
			ITC		:= (ITC_IO AND REAL_TO_BYTE(pow(2, IN_BitNumber))) <> 0;
		END_IF
	END_IF

	IF VAR_OldPage <> HMI_Page.PageNum THEN
		VAR_PageSwitch	:= TRUE;
	END_IF

	IF (Index = (VAR_ProgressiveId + 16 * HMI_Page.PageNum)) AND IN_Visibility THEN
		IF VAR_PageSwitch THEN
			IF IN_IOType THEN
				HMI_Data.DigitalOut[VAR_ProgressiveId].Auto	:= VAR_Auto;
				HMI_Data.DigitalOut[VAR_ProgressiveId].Man	:= VAR_Man;
			ELSE
				HMI_Data.DigitalIn[VAR_ProgressiveId].Auto	:= VAR_Auto;
				HMI_Data.DigitalIn[VAR_ProgressiveId].Man	:= VAR_Man;
			END_IF
			VAR_PageSwitch	:= FALSE;
		END_IF

		IF IN_IOType THEN
			HMI_Data.DigitalOut[VAR_ProgressiveId].Visibility	:= IN_Visibility;
			HMI_Data.DigitalOut[VAR_ProgressiveId].Enable		:= NOT IN_ReadOnly AND NOT IN_HMIAutoForce;
			HMI_Data.DigitalOut[VAR_ProgressiveId].LampState	:= (ITC_IO AND REAL_TO_BYTE(pow(2, IN_BitNumber))) <> 0;
			HMI_Data.DigitalOut[VAR_ProgressiveId].Wait			:= IN_Wait;
			HMI_Data.DigitalOut[VAR_ProgressiveId].Alarm		:= IN_Alarm;
			HMI_Data.DigitalOut[VAR_ProgressiveId].Description	:= IN_Description;

			IF EDGEPOS(HMI_Data.DigitalOut[VAR_ProgressiveId].Auto) THEN
				HMI_Data.DigitalOut[VAR_ProgressiveId].Man := FALSE;
			ELSIF EDGEPOS(HMI_Data.DigitalOut[VAR_ProgressiveId].Man) THEN
				HMI_Data.DigitalOut[VAR_ProgressiveId].Auto := FALSE;
			END_IF

			IF IN_ReadOnly OR IN_HMIAutoForce THEN
				HMI_Data.DigitalOut[VAR_ProgressiveId].Auto	:= TRUE;
				HMI_Data.DigitalOut[VAR_ProgressiveId].Man	:= FALSE;
			END_IF

			VAR_Auto	:= HMI_Data.DigitalOut[VAR_ProgressiveId].Auto;
			VAR_Man		:= HMI_Data.DigitalOut[VAR_ProgressiveId].Man;
		ELSE
			HMI_Data.DigitalIn[VAR_ProgressiveId].Visibility	:= IN_Visibility;
			HMI_Data.DigitalIn[VAR_ProgressiveId].Enable		:= NOT IN_ReadOnly AND NOT IN_HMIAutoForce;
			HMI_Data.DigitalIn[VAR_ProgressiveId].LampState 	:= ITC;
			HMI_Data.DigitalIn[VAR_ProgressiveId].Wait			:= IN_Wait;
			HMI_Data.DigitalIn[VAR_ProgressiveId].Alarm			:= IN_Alarm;
			HMI_Data.DigitalIn[VAR_ProgressiveId].Description	:= IN_Description;

			IF EDGEPOS(HMI_Data.DigitalIn[VAR_ProgressiveId].Auto) THEN
				HMI_Data.DigitalIn[VAR_ProgressiveId].Man := FALSE;
			ELSIF EDGEPOS(HMI_Data.DigitalIn[VAR_ProgressiveId].Man) THEN
				HMI_Data.DigitalIn[VAR_ProgressiveId].Auto := FALSE;
			END_IF

			IF IN_ReadOnly OR IN_HMIAutoForce THEN
				HMI_Data.DigitalIn[VAR_ProgressiveId].Auto	:= TRUE;
				HMI_Data.DigitalIn[VAR_ProgressiveId].Man	:= FALSE;
			END_IF

			VAR_Auto	:= HMI_Data.DigitalIn[VAR_ProgressiveId].Auto;
			VAR_Man		:= HMI_Data.DigitalIn[VAR_ProgressiveId].Man;
		END_IF
	ELSIF (Index < (VAR_ProgressiveId + 16 * HMI_Page.PageNum)) THEN
		IF IN_IOType THEN
			HMI_Data.DigitalOut[VAR_ProgressiveId].Visibility	:= FALSE;
		ELSE
			HMI_Data.DigitalIn[VAR_ProgressiveId].Visibility	:= FALSE;
		END_IF
	END_IF

	VAR_OldPage := HMI_Page.PageNum;

	HMI_Data.ManActive	:= NOT VAR_Auto OR HMI_Data.ManActive;

	IF (Index > (16 + 16 * HMI_Page.PageNum)) AND IN_Visibility THEN
		HMI_Data.PageUp.Enable := TRUE;
	END_IF

	IF HMI_Page.PageNum <> 0 THEN
		HMI_Data.PageDown.Enable := TRUE;
	END_IF

	OUT_Man			:= NOT VAR_Auto;
	OUT_ManValue	:= VAR_Man;
	Index			:= Index + 1;
END_FUNCTION_BLOCK

FUNCTION_BLOCK FB_HMI_ITC_DigitalUsint
	VAR_ProgressiveId := INT_TO_UINT(FC_ReminderShift(UINT_TO_INT(Index), 16, 0));

	IF IN_ReadOnly OR IN_HMIAutoForce THEN
		VAR_Auto	:= TRUE;
		VAR_Man		:= FALSE;
	END_IF

	IF IN_IOType THEN
		FOR VAR_BitIndex := 0 TO 7 DO
			IF VAR_BitIndex = INT_TO_USINT(IN_BitNumber) THEN
				IF NOT VAR_Auto THEN
					VAR_BitArray[VAR_BitIndex] := VAR_Man;
				ELSE
					VAR_BitArray[VAR_BitIndex] := ITC;
				END_IF
			ELSE
				VAR_BitArray[VAR_BitIndex] := (ITC_IO AND REAL_TO_USINT(pow(2, VAR_BitIndex))) <> 0;
			END_IF
		END_FOR

		ITC_IO	:= 0;

		FOR VAR_BitIndex := 0 TO 7 DO
			ITC_IO	:= ITC_IO OR UINT_TO_USINT(((REAL_TO_UINT(pow(2, VAR_BitIndex))) * VAR_BitArray[VAR_BitIndex]));
		END_FOR
	ELSE
		IF NOT VAR_Auto THEN
			ITC		:= VAR_Man;
		ELSE
			ITC		:= (ITC_IO AND REAL_TO_USINT(pow(2, IN_BitNumber))) <> 0;
		END_IF
	END_IF

	IF VAR_OldPage <> HMI_Page.PageNum THEN
		VAR_PageSwitch	:= TRUE;
	END_IF

	IF (Index = (VAR_ProgressiveId + 16 * HMI_Page.PageNum(*VAR_OldPage*))) AND IN_Visibility THEN
		IF VAR_PageSwitch THEN
			IF IN_IOType THEN
				HMI_Data.DigitalOut[VAR_ProgressiveId].Auto	:= VAR_Auto;
				HMI_Data.DigitalOut[VAR_ProgressiveId].Man	:= VAR_Man;
			ELSE
				HMI_Data.DigitalIn[VAR_ProgressiveId].Auto	:= VAR_Auto;
				HMI_Data.DigitalIn[VAR_ProgressiveId].Man	:= VAR_Man;
			END_IF
			VAR_PageSwitch	:= FALSE;
		END_IF

		IF IN_IOType THEN
			HMI_Data.DigitalOut[VAR_ProgressiveId].Visibility	:= IN_Visibility;
			HMI_Data.DigitalOut[VAR_ProgressiveId].Enable		:= NOT IN_ReadOnly AND NOT IN_HMIAutoForce;
			HMI_Data.DigitalOut[VAR_ProgressiveId].LampState	:= (ITC_IO AND REAL_TO_USINT(pow(2, IN_BitNumber))) <> 0;
			HMI_Data.DigitalOut[VAR_ProgressiveId].Wait			:= IN_Wait;
			HMI_Data.DigitalOut[VAR_ProgressiveId].Alarm		:= IN_Alarm;
			HMI_Data.DigitalOut[VAR_ProgressiveId].Description	:= IN_Description;

			IF EDGEPOS(HMI_Data.DigitalOut[VAR_ProgressiveId].Auto) THEN
				HMI_Data.DigitalOut[VAR_ProgressiveId].Man := FALSE;
				VAR_Man		:= FALSE;
			ELSIF EDGEPOS(HMI_Data.DigitalOut[VAR_ProgressiveId].Man) THEN
				HMI_Data.DigitalOut[VAR_ProgressiveId].Auto := FALSE;
				VAR_Auto	:= FALSE;
			END_IF

			IF IN_ReadOnly OR IN_HMIAutoForce THEN
				HMI_Data.DigitalOut[VAR_ProgressiveId].Auto	:= TRUE;
				HMI_Data.DigitalOut[VAR_ProgressiveId].Man	:= FALSE;
			END_IF

			VAR_Auto	:= HMI_Data.DigitalOut[VAR_ProgressiveId].Auto;
			VAR_Man		:= HMI_Data.DigitalOut[VAR_ProgressiveId].Man;
		ELSE
			HMI_Data.DigitalIn[VAR_ProgressiveId].Visibility	:= IN_Visibility;
			HMI_Data.DigitalIn[VAR_ProgressiveId].Enable		:= NOT IN_ReadOnly AND NOT IN_HMIAutoForce;
			HMI_Data.DigitalIn[VAR_ProgressiveId].LampState 	:= ITC;
			HMI_Data.DigitalIn[VAR_ProgressiveId].Wait			:= IN_Wait;
			HMI_Data.DigitalIn[VAR_ProgressiveId].Alarm			:= IN_Alarm;
			HMI_Data.DigitalIn[VAR_ProgressiveId].Description	:= IN_Description;

			IF EDGEPOS(HMI_Data.DigitalIn[VAR_ProgressiveId].Auto) THEN
				HMI_Data.DigitalIn[VAR_ProgressiveId].Man := FALSE;
			ELSIF EDGEPOS(HMI_Data.DigitalIn[VAR_ProgressiveId].Man) THEN
				HMI_Data.DigitalIn[VAR_ProgressiveId].Auto := FALSE;
			END_IF

			IF IN_ReadOnly OR IN_HMIAutoForce THEN
				HMI_Data.DigitalIn[VAR_ProgressiveId].Auto	:= TRUE;
				HMI_Data.DigitalIn[VAR_ProgressiveId].Man	:= FALSE;
			END_IF

			VAR_Auto	:= HMI_Data.DigitalIn[VAR_ProgressiveId].Auto;
			VAR_Man		:= HMI_Data.DigitalIn[VAR_ProgressiveId].Man;
		END_IF
	ELSIF (Index < (VAR_ProgressiveId + 16 * HMI_Page.PageNum(*VAR_OldPage*))) THEN
		IF IN_IOType THEN
			HMI_Data.DigitalOut[VAR_ProgressiveId].Visibility	:= FALSE;
		ELSE
			HMI_Data.DigitalIn[VAR_ProgressiveId].Visibility	:= FALSE;
		END_IF
	END_IF

	VAR_OldPage := HMI_Page.PageNum;

	HMI_Data.ManActive	:= NOT VAR_Auto OR HMI_Data.ManActive;

	IF (Index > (16 + 16 * HMI_Page.PageNum)) AND IN_Visibility THEN
		HMI_Data.PageUp.Enable := TRUE;
	END_IF

	IF HMI_Page.PageNum <> 0 THEN
		HMI_Data.PageDown.Enable := TRUE;
	END_IF

	OUT_Man			:= NOT VAR_Auto;
	OUT_ManValue	:= VAR_Man;
	Index			:= Index + 1;
END_FUNCTION_BLOCK

FUNCTION_BLOCK FB_HMI_ITC_DigitalInt
	VAR_ProgressiveId := INT_TO_UINT(FC_ReminderShift(UINT_TO_INT(Index), 16, 0));

	IF IN_ReadOnly OR IN_HMIAutoForce THEN
		VAR_Auto	:= TRUE;
		VAR_Man		:= FALSE;
	END_IF

	IF IN_IOType THEN
		FOR VAR_BitIndex := 0 TO 15 DO
			IF VAR_BitIndex = INT_TO_USINT(IN_BitNumber) THEN
				IF NOT VAR_Auto THEN
					VAR_BitArray[VAR_BitIndex] := VAR_Man;
				ELSE
					VAR_BitArray[VAR_BitIndex] := ITC;
				END_IF
			ELSE
				VAR_BitArray[VAR_BitIndex] := (ITC_IO AND REAL_TO_INT(pow(2, VAR_BitIndex))) <> 0;
			END_IF
		END_FOR

		ITC_IO	:= 0;

		FOR VAR_BitIndex := 0 TO 15 DO
			ITC_IO	:= ITC_IO OR UINT_TO_INT(((REAL_TO_UINT(pow(2, VAR_BitIndex))) * VAR_BitArray[VAR_BitIndex]));
		END_FOR
	ELSE
		IF NOT VAR_Auto THEN
			ITC		:= VAR_Man;
		ELSE
			ITC		:= (ITC_IO AND REAL_TO_INT(pow(2, IN_BitNumber))) <> 0;
		END_IF
	END_IF

	IF VAR_OldPage <> HMI_Page.PageNum THEN
		VAR_PageSwitch	:= TRUE;
	END_IF

	IF (Index = (VAR_ProgressiveId + 16 * HMI_Page.PageNum)) AND IN_Visibility THEN
		IF VAR_PageSwitch THEN
			IF IN_IOType THEN
				HMI_Data.DigitalOut[VAR_ProgressiveId].Auto	:= VAR_Auto;
				HMI_Data.DigitalOut[VAR_ProgressiveId].Man	:= VAR_Man;
			ELSE
				HMI_Data.DigitalIn[VAR_ProgressiveId].Auto	:= VAR_Auto;
				HMI_Data.DigitalIn[VAR_ProgressiveId].Man	:= VAR_Man;
			END_IF
			VAR_PageSwitch	:= FALSE;
		END_IF

		IF IN_IOType THEN
			HMI_Data.DigitalOut[VAR_ProgressiveId].Visibility	:= IN_Visibility;
			HMI_Data.DigitalOut[VAR_ProgressiveId].Enable		:= NOT IN_ReadOnly AND NOT IN_HMIAutoForce;
			HMI_Data.DigitalOut[VAR_ProgressiveId].LampState	:= (ITC_IO AND REAL_TO_INT(pow(2, IN_BitNumber))) <> 0;
			HMI_Data.DigitalOut[VAR_ProgressiveId].Wait			:= IN_Wait;
			HMI_Data.DigitalOut[VAR_ProgressiveId].Alarm		:= IN_Alarm;
			HMI_Data.DigitalOut[VAR_ProgressiveId].Description	:= IN_Description;

			IF EDGEPOS(HMI_Data.DigitalOut[VAR_ProgressiveId].Auto) THEN
				HMI_Data.DigitalOut[VAR_ProgressiveId].Man := FALSE;
			ELSIF EDGEPOS(HMI_Data.DigitalOut[VAR_ProgressiveId].Man) THEN
				HMI_Data.DigitalOut[VAR_ProgressiveId].Auto := FALSE;
			END_IF

			VAR_Auto	:= HMI_Data.DigitalOut[VAR_ProgressiveId].Auto;
			VAR_Man		:= HMI_Data.DigitalOut[VAR_ProgressiveId].Man;
		ELSE
			HMI_Data.DigitalIn[VAR_ProgressiveId].Visibility	:= IN_Visibility;
			HMI_Data.DigitalIn[VAR_ProgressiveId].Enable		:= NOT IN_ReadOnly AND NOT IN_HMIAutoForce;
			HMI_Data.DigitalIn[VAR_ProgressiveId].LampState 	:= ITC;
			HMI_Data.DigitalIn[VAR_ProgressiveId].Wait			:= IN_Wait;
			HMI_Data.DigitalIn[VAR_ProgressiveId].Alarm			:= IN_Alarm;
			HMI_Data.DigitalIn[VAR_ProgressiveId].Description	:= IN_Description;

			IF EDGEPOS(HMI_Data.DigitalIn[VAR_ProgressiveId].Auto) THEN
				HMI_Data.DigitalIn[VAR_ProgressiveId].Man := FALSE;
			ELSIF EDGEPOS(HMI_Data.DigitalIn[VAR_ProgressiveId].Man) THEN
				HMI_Data.DigitalIn[VAR_ProgressiveId].Auto := FALSE;
			END_IF

			VAR_Auto	:= HMI_Data.DigitalIn[VAR_ProgressiveId].Auto;
			VAR_Man		:= HMI_Data.DigitalIn[VAR_ProgressiveId].Man;
		END_IF
	ELSIF (Index < (VAR_ProgressiveId + 16 * HMI_Page.PageNum)) THEN
		IF IN_IOType THEN
			HMI_Data.DigitalOut[VAR_ProgressiveId].Visibility	:= FALSE;
		ELSE
			HMI_Data.DigitalIn[VAR_ProgressiveId].Visibility	:= FALSE;
		END_IF
	END_IF

	VAR_OldPage := HMI_Page.PageNum;

	HMI_Data.ManActive	:= NOT VAR_Auto OR HMI_Data.ManActive;

	IF (Index > (16 + 16 * HMI_Page.PageNum)) AND IN_Visibility THEN
		HMI_Data.PageUp.Enable := TRUE;
	END_IF

	IF HMI_Page.PageNum <> 0 THEN
		HMI_Data.PageDown.Enable := TRUE;
	END_IF

	OUT_Man			:= NOT VAR_Auto;
	OUT_ManValue	:= VAR_Man;
	Index			:= Index + 1;
END_FUNCTION_BLOCK

FUNCTION_BLOCK FB_HMI_ITC_AnalogByte
	VAR_ProgressiveId := INT_TO_UINT(FC_ReminderShift(UINT_TO_INT(Index), 4, 0));

	IF IN_ReadOnly OR IN_HMIAutoForce THEN
		VAR_Man		:= FALSE;
	END_IF

	IF IN_IOType THEN
		ITC_IO 		:= SEL(VAR_Man, ITC, VAR_ManValue);
	ELSE
		ITC 		:= SEL(VAR_Man, ITC_IO, VAR_ManValue);
	END_IF

	IF VAR_OldPage <> HMI_Page.PageNum THEN
		VAR_PageSwitch	:= TRUE;
	END_IF

	IF (Index = (VAR_ProgressiveId + 4 * HMI_Page.PageNum)) AND IN_Visibility THEN
		IF VAR_PageSwitch THEN
			IF IN_IOType THEN
				HMI_Data.AnalogOut[VAR_ProgressiveId].Man		:= VAR_Man;
				HMI_Data.AnalogOut[VAR_ProgressiveId].PV_Man	:= BYTE_TO_REAL(VAR_ManValue);
			ELSE
				HMI_Data.AnalogIn[VAR_ProgressiveId].Man		:= VAR_Man;
				HMI_Data.AnalogIn[VAR_ProgressiveId].PV_Man		:= BYTE_TO_REAL(VAR_ManValue);
			END_IF
			VAR_PageSwitch	:= FALSE;
		END_IF

		IF IN_IOType THEN
			HMI_Data.AnalogOut[VAR_ProgressiveId].Visibility	:= IN_Visibility;
			HMI_Data.AnalogOut[VAR_ProgressiveId].Enable		:= NOT IN_ReadOnly AND NOT IN_HMIAutoForce;
			HMI_Data.AnalogOut[VAR_ProgressiveId].PV			:= BYTE_TO_REAL(ITC_IO);
			HMI_Data.AnalogOut[VAR_ProgressiveId].Wait			:= IN_Wait;
			HMI_Data.AnalogOut[VAR_ProgressiveId].Description	:= IN_Description;
			HMI_Data.AnalogOut[VAR_ProgressiveId].Unit			:= IN_Unit;
			HMI_Data.AnalogOut[VAR_ProgressiveId].MaxValue		:= IN_MaxValue;
			HMI_Data.AnalogOut[VAR_ProgressiveId].MinValue		:= IN_MinValue;

			VAR_Man			:= HMI_Data.AnalogOut[VAR_ProgressiveId].Man;
			VAR_ManValue	:= REAL_TO_BYTE(HMI_Data.AnalogOut[VAR_ProgressiveId].PV_Man);
		ELSE
			HMI_Data.AnalogIn[VAR_ProgressiveId].Visibility		:= IN_Visibility;
			HMI_Data.AnalogIn[VAR_ProgressiveId].Enable			:= NOT IN_ReadOnly AND NOT IN_HMIAutoForce;
			HMI_Data.AnalogIn[VAR_ProgressiveId].PV				:= BYTE_TO_REAL(ITC);
			HMI_Data.AnalogIn[VAR_ProgressiveId].Wait			:= IN_Wait;
			HMI_Data.AnalogIn[VAR_ProgressiveId].Description	:= IN_Description;
			HMI_Data.AnalogIn[VAR_ProgressiveId].Unit			:= IN_Unit;
			HMI_Data.AnalogIn[VAR_ProgressiveId].MaxValue		:= IN_MaxValue;
			HMI_Data.AnalogIn[VAR_ProgressiveId].MinValue		:= IN_MinValue;

			VAR_Man			:= HMI_Data.AnalogIn[VAR_ProgressiveId].Man;
			VAR_ManValue	:= REAL_TO_BYTE(HMI_Data.AnalogIn[VAR_ProgressiveId].PV_Man);
		END_IF
	ELSIF (Index < (VAR_ProgressiveId + 4 * HMI_Page.PageNum)) THEN
		IF IN_IOType THEN
			HMI_Data.AnalogOut[VAR_ProgressiveId].Visibility	:= FALSE;
		ELSE
			HMI_Data.AnalogIn[VAR_ProgressiveId].Visibility		:= FALSE;
		END_IF
	END_IF

	VAR_OldPage := HMI_Page.PageNum;

	HMI_Data.ManActive	:= VAR_Man OR HMI_Data.ManActive;

	IF (Index > (4 + 4 * HMI_Page.PageNum)) AND IN_Visibility THEN
		HMI_Data.PageUp.Enable := TRUE;
	END_IF

	IF HMI_Page.PageNum <> 0 THEN
		HMI_Data.PageDown.Enable := TRUE;
	END_IF

	OUT_Man			:= VAR_Man;
	OUT_ManValue	:= VAR_ManValue;
	Index			:= Index + 1;
END_FUNCTION_BLOCK

FUNCTION_BLOCK FB_HMI_ITC_AnalogUsint
	VAR_ProgressiveId := INT_TO_UINT(FC_ReminderShift(UINT_TO_INT(Index), 4, 0));

	IF IN_ReadOnly OR IN_HMIAutoForce THEN
		VAR_Man		:= FALSE;
	END_IF

	IF IN_IOType THEN
		ITC_IO 		:= SEL(VAR_Man, ITC, VAR_ManValue);
	ELSE
		ITC 		:= SEL(VAR_Man, ITC_IO, VAR_ManValue);
	END_IF

	IF VAR_OldPage <> HMI_Page.PageNum THEN
		VAR_PageSwitch	:= TRUE;
	END_IF

	IF (Index = (VAR_ProgressiveId + 4 * HMI_Page.PageNum)) AND IN_Visibility THEN
		IF VAR_PageSwitch THEN
			IF IN_IOType THEN
				HMI_Data.AnalogOut[VAR_ProgressiveId].Man		:= VAR_Man;
				HMI_Data.AnalogOut[VAR_ProgressiveId].PV_Man	:= USINT_TO_REAL(VAR_ManValue);
			ELSE
				HMI_Data.AnalogIn[VAR_ProgressiveId].Man		:= VAR_Man;
				HMI_Data.AnalogIn[VAR_ProgressiveId].PV_Man		:= USINT_TO_REAL(VAR_ManValue);
			END_IF
			VAR_PageSwitch	:= FALSE;
		END_IF

		IF IN_IOType THEN
			HMI_Data.AnalogOut[VAR_ProgressiveId].Visibility	:= IN_Visibility;
			HMI_Data.AnalogOut[VAR_ProgressiveId].Enable		:= NOT IN_ReadOnly AND NOT IN_HMIAutoForce;
			HMI_Data.AnalogOut[VAR_ProgressiveId].PV			:= USINT_TO_REAL(ITC_IO);
			HMI_Data.AnalogOut[VAR_ProgressiveId].Wait			:= IN_Wait;
			HMI_Data.AnalogOut[VAR_ProgressiveId].Description	:= IN_Description;
			HMI_Data.AnalogOut[VAR_ProgressiveId].Unit			:= IN_Unit;
			HMI_Data.AnalogOut[VAR_ProgressiveId].MaxValue		:= IN_MaxValue;
			HMI_Data.AnalogOut[VAR_ProgressiveId].MinValue		:= IN_MinValue;

			VAR_Man			:= HMI_Data.AnalogOut[VAR_ProgressiveId].Man;
			VAR_ManValue	:= REAL_TO_USINT(HMI_Data.AnalogOut[VAR_ProgressiveId].PV_Man);
		ELSE
			HMI_Data.AnalogIn[VAR_ProgressiveId].Visibility		:= IN_Visibility;
			HMI_Data.AnalogIn[VAR_ProgressiveId].Enable			:= NOT IN_ReadOnly AND NOT IN_HMIAutoForce;
			HMI_Data.AnalogIn[VAR_ProgressiveId].PV				:= USINT_TO_REAL(ITC);
			HMI_Data.AnalogIn[VAR_ProgressiveId].Wait			:= IN_Wait;
			HMI_Data.AnalogIn[VAR_ProgressiveId].Description	:= IN_Description;
			HMI_Data.AnalogIn[VAR_ProgressiveId].Unit			:= IN_Unit;
			HMI_Data.AnalogIn[VAR_ProgressiveId].MaxValue		:= IN_MaxValue;
			HMI_Data.AnalogIn[VAR_ProgressiveId].MinValue		:= IN_MinValue;

			VAR_Man			:= HMI_Data.AnalogIn[VAR_ProgressiveId].Man;
			VAR_ManValue	:= REAL_TO_USINT(HMI_Data.AnalogIn[VAR_ProgressiveId].PV_Man);
		END_IF
	ELSIF (Index < (VAR_ProgressiveId + 4 * HMI_Page.PageNum)) THEN
		IF IN_IOType THEN
			HMI_Data.AnalogOut[VAR_ProgressiveId].Visibility	:= FALSE;
		ELSE
			HMI_Data.AnalogIn[VAR_ProgressiveId].Visibility		:= FALSE;
		END_IF
	END_IF

	VAR_OldPage := HMI_Page.PageNum;

	HMI_Data.ManActive	:= VAR_Man OR HMI_Data.ManActive;

	IF (Index > (4 + 4 * HMI_Page.PageNum)) AND IN_Visibility THEN
		HMI_Data.PageUp.Enable := TRUE;
	END_IF

	IF HMI_Page.PageNum <> 0 THEN
		HMI_Data.PageDown.Enable := TRUE;
	END_IF

	OUT_Man			:= VAR_Man;
	OUT_ManValue	:= VAR_ManValue;
	Index			:= Index + 1;
END_FUNCTION_BLOCK

FUNCTION_BLOCK FB_HMI_ITC_AnalogInt
	VAR_ProgressiveId := INT_TO_UINT(FC_ReminderShift(UINT_TO_INT(Index), 4, 0));

	IF IN_ReadOnly OR IN_HMIAutoForce THEN
		VAR_Man		:= FALSE;
	END_IF

	IF IN_IOType THEN
		VAR_Value 	:= SEL(VAR_Man, ITC, VAR_ManValue);
		ITC_IO 		:= SEL(HMI_Data.ComSwap, VAR_Value, swapINT(VAR_Value));
	ELSE
		VAR_Value 	:= SEL(HMI_Data.ComSwap, ITC_IO, swapINT(ITC_IO));
		ITC 		:= SEL(VAR_Man, VAR_Value, VAR_ManValue);
	END_IF

	IF VAR_OldPage <> HMI_Page.PageNum THEN
		VAR_PageSwitch	:= TRUE;
	END_IF

	IF (Index = (VAR_ProgressiveId + 4 * HMI_Page.PageNum)) AND IN_Visibility THEN
		IF VAR_PageSwitch THEN
			IF IN_IOType THEN
				HMI_Data.AnalogOut[VAR_ProgressiveId].Man		:= VAR_Man;
				HMI_Data.AnalogOut[VAR_ProgressiveId].PV_Man	:= INT_TO_REAL(VAR_ManValue);
			ELSE
				HMI_Data.AnalogIn[VAR_ProgressiveId].Man		:= VAR_Man;
				HMI_Data.AnalogIn[VAR_ProgressiveId].PV_Man		:= INT_TO_REAL(VAR_ManValue);
			END_IF
			VAR_PageSwitch	:= FALSE;
		END_IF

		IF IN_IOType THEN
			HMI_Data.AnalogOut[VAR_ProgressiveId].Visibility	:= IN_Visibility;
			HMI_Data.AnalogOut[VAR_ProgressiveId].Enable		:= NOT IN_ReadOnly AND NOT IN_HMIAutoForce;
			HMI_Data.AnalogOut[VAR_ProgressiveId].PV			:= INT_TO_REAL(VAR_Value);
			HMI_Data.AnalogOut[VAR_ProgressiveId].Wait			:= IN_Wait;
			HMI_Data.AnalogOut[VAR_ProgressiveId].Description	:= IN_Description;
			HMI_Data.AnalogOut[VAR_ProgressiveId].Unit			:= IN_Unit;
			HMI_Data.AnalogOut[VAR_ProgressiveId].MaxValue		:= IN_MaxValue;
			HMI_Data.AnalogOut[VAR_ProgressiveId].MinValue		:= IN_MinValue;

			VAR_Man			:= HMI_Data.AnalogOut[VAR_ProgressiveId].Man;
			VAR_ManValue	:= REAL_TO_INT(HMI_Data.AnalogOut[VAR_ProgressiveId].PV_Man);
		ELSE
			HMI_Data.AnalogIn[VAR_ProgressiveId].Visibility		:= IN_Visibility;
			HMI_Data.AnalogIn[VAR_ProgressiveId].Enable			:= NOT IN_ReadOnly AND NOT IN_HMIAutoForce;
			HMI_Data.AnalogIn[VAR_ProgressiveId].PV				:= INT_TO_REAL(ITC);
			HMI_Data.AnalogIn[VAR_ProgressiveId].Wait			:= IN_Wait;
			HMI_Data.AnalogIn[VAR_ProgressiveId].Description	:= IN_Description;
			HMI_Data.AnalogIn[VAR_ProgressiveId].Unit			:= IN_Unit;
			HMI_Data.AnalogIn[VAR_ProgressiveId].MaxValue		:= IN_MaxValue;
			HMI_Data.AnalogIn[VAR_ProgressiveId].MinValue		:= IN_MinValue;

			VAR_Man			:= HMI_Data.AnalogIn[VAR_ProgressiveId].Man;
			VAR_ManValue	:= REAL_TO_INT(HMI_Data.AnalogIn[VAR_ProgressiveId].PV_Man);
		END_IF
	ELSIF (Index < (VAR_ProgressiveId + 4 * HMI_Page.PageNum)) THEN
		IF IN_IOType THEN
			HMI_Data.AnalogOut[VAR_ProgressiveId].Visibility	:= FALSE;
		ELSE
			HMI_Data.AnalogIn[VAR_ProgressiveId].Visibility		:= FALSE;
		END_IF
	END_IF

	VAR_OldPage := HMI_Page.PageNum;

	HMI_Data.ManActive	:= VAR_Man OR HMI_Data.ManActive;

	IF (Index > (4 + 4 * HMI_Page.PageNum)) AND IN_Visibility THEN
		HMI_Data.PageUp.Enable := TRUE;
	END_IF

	IF HMI_Page.PageNum <> 0 THEN
		HMI_Data.PageDown.Enable := TRUE;
	END_IF

	OUT_Man			:= VAR_Man;
	OUT_ManValue	:= VAR_ManValue;
	Index			:= Index + 1;
END_FUNCTION_BLOCK

FUNCTION_BLOCK FB_HMI_ITC_AnalogIntOverUsint
	VAR_ProgressiveId := INT_TO_UINT(FC_ReminderShift(UINT_TO_INT(Index), 4, 0));

	IF IN_ReadOnly OR IN_HMIAutoForce THEN
		VAR_Man		:= FALSE;
	END_IF

	IF IN_IOType THEN
		VAR_Value		:= SEL(VAR_Man, ITC, VAR_ManValue);
		VAR_RawValue	:= SEL(HMI_Data.ComSwap, VAR_Value, swapINT(VAR_Value));
		memcpy(ADR(ITC_IO), ADR(VAR_RawValue), SIZEOF(ITC));
	ELSE
		memcpy(ADR(VAR_RawValue), ADR(ITC_IO), SIZEOF(ITC));
		VAR_Value	:= SEL(HMI_Data.ComSwap, VAR_RawValue, swapINT(VAR_RawValue));
		ITC			:= SEL(VAR_Man, VAR_Value, VAR_ManValue);
	END_IF

	IF VAR_OldPage <> HMI_Page.PageNum THEN
		VAR_PageSwitch	:= TRUE;
	END_IF

	IF (Index = (VAR_ProgressiveId + 4 * HMI_Page.PageNum)) AND IN_Visibility THEN
		IF VAR_PageSwitch THEN
			IF IN_IOType THEN
				HMI_Data.AnalogOut[VAR_ProgressiveId].Man		:= VAR_Man;
				HMI_Data.AnalogOut[VAR_ProgressiveId].PV_Man	:= INT_TO_REAL(VAR_ManValue);
			ELSE
				HMI_Data.AnalogIn[VAR_ProgressiveId].Man		:= VAR_Man;
				HMI_Data.AnalogIn[VAR_ProgressiveId].PV_Man		:= INT_TO_REAL(VAR_ManValue);
			END_IF
			VAR_PageSwitch	:= FALSE;
		END_IF

		IF IN_IOType THEN
			HMI_Data.AnalogOut[VAR_ProgressiveId].Visibility	:= IN_Visibility;
			HMI_Data.AnalogOut[VAR_ProgressiveId].Enable		:= NOT IN_ReadOnly AND NOT IN_HMIAutoForce;
			HMI_Data.AnalogOut[VAR_ProgressiveId].PV			:= INT_TO_REAL(VAR_Value);
			HMI_Data.AnalogOut[VAR_ProgressiveId].Wait			:= IN_Wait;
			HMI_Data.AnalogOut[VAR_ProgressiveId].Description	:= IN_Description;
			HMI_Data.AnalogOut[VAR_ProgressiveId].Unit			:= IN_Unit;
			HMI_Data.AnalogOut[VAR_ProgressiveId].MaxValue		:= IN_MaxValue;
			HMI_Data.AnalogOut[VAR_ProgressiveId].MinValue		:= IN_MinValue;

			VAR_Man			:= HMI_Data.AnalogOut[VAR_ProgressiveId].Man;
			VAR_ManValue	:= REAL_TO_INT(HMI_Data.AnalogOut[VAR_ProgressiveId].PV_Man);
		ELSE
			HMI_Data.AnalogIn[VAR_ProgressiveId].Visibility		:= IN_Visibility;
			HMI_Data.AnalogIn[VAR_ProgressiveId].Enable			:= NOT IN_ReadOnly AND NOT IN_HMIAutoForce;
			HMI_Data.AnalogIn[VAR_ProgressiveId].PV				:= INT_TO_REAL(ITC);
			HMI_Data.AnalogIn[VAR_ProgressiveId].Wait			:= IN_Wait;
			HMI_Data.AnalogIn[VAR_ProgressiveId].Description	:= IN_Description;
			HMI_Data.AnalogIn[VAR_ProgressiveId].Unit			:= IN_Unit;
			HMI_Data.AnalogIn[VAR_ProgressiveId].MaxValue		:= IN_MaxValue;
			HMI_Data.AnalogIn[VAR_ProgressiveId].MinValue		:= IN_MinValue;

			VAR_Man			:= HMI_Data.AnalogIn[VAR_ProgressiveId].Man;
			VAR_ManValue	:= REAL_TO_INT(HMI_Data.AnalogIn[VAR_ProgressiveId].PV_Man);
		END_IF
	ELSIF (Index < (VAR_ProgressiveId + 4 * HMI_Page.PageNum)) THEN
		IF IN_IOType THEN
			HMI_Data.AnalogOut[VAR_ProgressiveId].Visibility	:= FALSE;
		ELSE
			HMI_Data.AnalogIn[VAR_ProgressiveId].Visibility		:= FALSE;
		END_IF
	END_IF

	VAR_OldPage := HMI_Page.PageNum;

	HMI_Data.ManActive	:= VAR_Man OR HMI_Data.ManActive;

	IF (Index > (4 + 4 * HMI_Page.PageNum)) AND IN_Visibility THEN
		HMI_Data.PageUp.Enable := TRUE;
	END_IF

	IF HMI_Page.PageNum <> 0 THEN
		HMI_Data.PageDown.Enable := TRUE;
	END_IF

	OUT_Man			:= VAR_Man;
	OUT_ManValue	:= VAR_ManValue;
	Index			:= Index + 1;
END_FUNCTION_BLOCK

FUNCTION_BLOCK FB_HMI_ITC_AnalogUintOverUsint
	VAR_ProgressiveId := INT_TO_UINT(FC_ReminderShift(UINT_TO_INT(Index), 4, 0));

	IF IN_ReadOnly OR IN_HMIAutoForce THEN
		VAR_Man		:= FALSE;
	END_IF

	IF IN_IOType THEN
		VAR_Value		:= SEL(VAR_Man, ITC, VAR_ManValue);
		VAR_RawValue	:= SEL(HMI_Data.ComSwap, VAR_Value, swapINT(VAR_Value));
		memcpy(ADR(ITC_IO), ADR(VAR_RawValue), SIZEOF(ITC));
	ELSE
		memcpy(ADR(VAR_RawValue), ADR(ITC_IO), SIZEOF(ITC));
		VAR_Value	:= SEL(HMI_Data.ComSwap, VAR_RawValue, swapINT(VAR_RawValue));
		ITC			:= SEL(VAR_Man, VAR_Value, VAR_ManValue);
	END_IF

	IF VAR_OldPage <> HMI_Page.PageNum THEN
		VAR_PageSwitch	:= TRUE;
	END_IF

	IF (Index = (VAR_ProgressiveId + 4 * HMI_Page.PageNum)) AND IN_Visibility THEN
		IF VAR_PageSwitch THEN
			IF IN_IOType THEN
				HMI_Data.AnalogOut[VAR_ProgressiveId].Man		:= VAR_Man;
				HMI_Data.AnalogOut[VAR_ProgressiveId].PV_Man	:= INT_TO_REAL(VAR_ManValue);
			ELSE
				HMI_Data.AnalogIn[VAR_ProgressiveId].Man		:= VAR_Man;
				HMI_Data.AnalogIn[VAR_ProgressiveId].PV_Man		:= INT_TO_REAL(VAR_ManValue);
			END_IF
			VAR_PageSwitch	:= FALSE;
		END_IF

		IF IN_IOType THEN
			HMI_Data.AnalogOut[VAR_ProgressiveId].Visibility	:= IN_Visibility;
			HMI_Data.AnalogOut[VAR_ProgressiveId].Enable		:= NOT IN_ReadOnly AND NOT IN_HMIAutoForce;
			HMI_Data.AnalogOut[VAR_ProgressiveId].PV			:= INT_TO_REAL(VAR_Value);
			HMI_Data.AnalogOut[VAR_ProgressiveId].Wait			:= IN_Wait;
			HMI_Data.AnalogOut[VAR_ProgressiveId].Description	:= IN_Description;
			HMI_Data.AnalogOut[VAR_ProgressiveId].Unit			:= IN_Unit;
			HMI_Data.AnalogOut[VAR_ProgressiveId].MaxValue		:= IN_MaxValue;
			HMI_Data.AnalogOut[VAR_ProgressiveId].MinValue		:= IN_MinValue;

			VAR_Man			:= HMI_Data.AnalogOut[VAR_ProgressiveId].Man;
			VAR_ManValue	:= REAL_TO_INT(HMI_Data.AnalogOut[VAR_ProgressiveId].PV_Man);
		ELSE
			HMI_Data.AnalogIn[VAR_ProgressiveId].Visibility		:= IN_Visibility;
			HMI_Data.AnalogIn[VAR_ProgressiveId].Enable			:= NOT IN_ReadOnly AND NOT IN_HMIAutoForce;
			HMI_Data.AnalogIn[VAR_ProgressiveId].PV				:= INT_TO_REAL(ITC);
			HMI_Data.AnalogIn[VAR_ProgressiveId].Wait			:= IN_Wait;
			HMI_Data.AnalogIn[VAR_ProgressiveId].Description	:= IN_Description;
			HMI_Data.AnalogIn[VAR_ProgressiveId].Unit			:= IN_Unit;
			HMI_Data.AnalogIn[VAR_ProgressiveId].MaxValue		:= IN_MaxValue;
			HMI_Data.AnalogIn[VAR_ProgressiveId].MinValue		:= IN_MinValue;

			VAR_Man			:= HMI_Data.AnalogIn[VAR_ProgressiveId].Man;
			VAR_ManValue	:= REAL_TO_INT(HMI_Data.AnalogIn[VAR_ProgressiveId].PV_Man);
		END_IF
	ELSIF (Index < (VAR_ProgressiveId + 4 * HMI_Page.PageNum)) THEN
		IF IN_IOType THEN
			HMI_Data.AnalogOut[VAR_ProgressiveId].Visibility	:= FALSE;
		ELSE
			HMI_Data.AnalogIn[VAR_ProgressiveId].Visibility		:= FALSE;
		END_IF
	END_IF

	VAR_OldPage := HMI_Page.PageNum;

	HMI_Data.ManActive	:= VAR_Man OR HMI_Data.ManActive;

	IF (Index > (4 + 4 * HMI_Page.PageNum)) AND IN_Visibility THEN
		HMI_Data.PageUp.Enable := TRUE;
	END_IF

	IF HMI_Page.PageNum <> 0 THEN
		HMI_Data.PageDown.Enable := TRUE;
	END_IF

	OUT_Man			:= VAR_Man;
	OUT_ManValue	:= VAR_ManValue;
	Index			:= Index + 1;
END_FUNCTION_BLOCK

FUNCTION_BLOCK FB_HMI_ITC_AnalogDInt
	VAR_ProgressiveId := INT_TO_UINT(FC_ReminderShift(UINT_TO_INT(Index), 4, 0));

	IF IN_ReadOnly OR IN_HMIAutoForce THEN
		VAR_Man		:= FALSE;
	END_IF

	IF IN_IOType THEN
		VAR_Value	:= SEL(VAR_Man, ITC, VAR_ManValue);
		ITC_IO		:= SEL(HMI_Data.ComSwap, VAR_Value, swapDINT(VAR_Value));
	ELSE
		VAR_Value	:= SEL(HMI_Data.ComSwap, ITC_IO, swapDINT(ITC_IO));
		ITC			:= SEL(VAR_Man, VAR_Value, VAR_ManValue);
	END_IF

	IF VAR_OldPage <> HMI_Page.PageNum THEN
		VAR_PageSwitch	:= TRUE;
	END_IF

	IF (Index = (VAR_ProgressiveId + 4 * HMI_Page.PageNum)) AND IN_Visibility THEN
		IF VAR_PageSwitch THEN
			IF IN_IOType THEN
				HMI_Data.AnalogOut[VAR_ProgressiveId].Man		:= VAR_Man;
				HMI_Data.AnalogOut[VAR_ProgressiveId].PV_Man	:= DINT_TO_REAL(VAR_ManValue);
			ELSE
				HMI_Data.AnalogIn[VAR_ProgressiveId].Man		:= VAR_Man;
				HMI_Data.AnalogIn[VAR_ProgressiveId].PV_Man		:= DINT_TO_REAL(VAR_ManValue);
			END_IF
			VAR_PageSwitch	:= FALSE;
		END_IF

		IF IN_IOType THEN
			HMI_Data.AnalogOut[VAR_ProgressiveId].Visibility	:= IN_Visibility;
			HMI_Data.AnalogOut[VAR_ProgressiveId].Enable		:= NOT IN_ReadOnly AND NOT IN_HMIAutoForce;
			HMI_Data.AnalogOut[VAR_ProgressiveId].PV			:= DINT_TO_REAL(VAR_Value);
			HMI_Data.AnalogOut[VAR_ProgressiveId].Wait			:= IN_Wait;
			HMI_Data.AnalogOut[VAR_ProgressiveId].Description	:= IN_Description;
			HMI_Data.AnalogOut[VAR_ProgressiveId].Unit			:= IN_Unit;
			HMI_Data.AnalogOut[VAR_ProgressiveId].MaxValue		:= IN_MaxValue;
			HMI_Data.AnalogOut[VAR_ProgressiveId].MinValue		:= IN_MinValue;

			VAR_Man			:= HMI_Data.AnalogOut[VAR_ProgressiveId].Man;
			VAR_ManValue	:= REAL_TO_INT(HMI_Data.AnalogOut[VAR_ProgressiveId].PV_Man);
		ELSE
			HMI_Data.AnalogIn[VAR_ProgressiveId].Visibility		:= IN_Visibility;
			HMI_Data.AnalogIn[VAR_ProgressiveId].Enable			:= NOT IN_ReadOnly AND NOT IN_HMIAutoForce;
			HMI_Data.AnalogIn[VAR_ProgressiveId].PV				:= DINT_TO_REAL(ITC);
			HMI_Data.AnalogIn[VAR_ProgressiveId].Wait			:= IN_Wait;
			HMI_Data.AnalogIn[VAR_ProgressiveId].Description	:= IN_Description;
			HMI_Data.AnalogIn[VAR_ProgressiveId].Unit			:= IN_Unit;
			HMI_Data.AnalogIn[VAR_ProgressiveId].MaxValue		:= IN_MaxValue;
			HMI_Data.AnalogIn[VAR_ProgressiveId].MinValue		:= IN_MinValue;

			VAR_Man			:= HMI_Data.AnalogIn[VAR_ProgressiveId].Man;
			VAR_ManValue	:= REAL_TO_INT(HMI_Data.AnalogIn[VAR_ProgressiveId].PV_Man);
		END_IF
	ELSIF (Index < (VAR_ProgressiveId + 4 * HMI_Page.PageNum)) THEN
		IF IN_IOType THEN
			HMI_Data.AnalogOut[VAR_ProgressiveId].Visibility	:= FALSE;
		ELSE
			HMI_Data.AnalogIn[VAR_ProgressiveId].Visibility		:= FALSE;
		END_IF
	END_IF

	VAR_OldPage := HMI_Page.PageNum;

	HMI_Data.ManActive	:= VAR_Man OR HMI_Data.ManActive;

	IF (Index > (4 + 4 * HMI_Page.PageNum)) AND IN_Visibility THEN
		HMI_Data.PageUp.Enable := TRUE;
	END_IF

	IF HMI_Page.PageNum <> 0 THEN
		HMI_Data.PageDown.Enable := TRUE;
	END_IF

	OUT_Man			:= VAR_Man;
	OUT_ManValue	:= VAR_ManValue;
	Index	:= Index + 1;
END_FUNCTION_BLOCK

FUNCTION_BLOCK FB_HMI_ITC_AnalogUdint
	VAR_ProgressiveId := INT_TO_UINT(FC_ReminderShift(UINT_TO_INT(Index), 4, 0));

	IF IN_ReadOnly OR IN_HMIAutoForce THEN
		VAR_Man		:= FALSE;
	END_IF

	IF IN_IOType THEN
		VAR_Value	:= SEL(VAR_Man, ITC, VAR_ManValue);
		ITC_IO		:= SEL(HMI_Data.ComSwap, VAR_Value, swapUDINT(VAR_Value));
	ELSE
		VAR_Value	:= SEL(HMI_Data.ComSwap, ITC_IO, swapUDINT(ITC_IO));
		ITC			:= SEL(VAR_Man, VAR_Value, VAR_ManValue);
	END_IF

	IF VAR_OldPage <> HMI_Page.PageNum THEN
		VAR_PageSwitch	:= TRUE;
	END_IF

	IF (Index = (VAR_ProgressiveId + 4 * HMI_Page.PageNum)) AND IN_Visibility THEN
		IF VAR_PageSwitch THEN
			IF IN_IOType THEN
				HMI_Data.AnalogOut[VAR_ProgressiveId].Man		:= VAR_Man;
				HMI_Data.AnalogOut[VAR_ProgressiveId].PV_Man	:= UDINT_TO_REAL(VAR_ManValue);
			ELSE
				HMI_Data.AnalogIn[VAR_ProgressiveId].Man		:= VAR_Man;
				HMI_Data.AnalogIn[VAR_ProgressiveId].PV_Man		:= UDINT_TO_REAL(VAR_ManValue);
			END_IF
			VAR_PageSwitch	:= FALSE;
		END_IF

		IF IN_IOType THEN
			HMI_Data.AnalogOut[VAR_ProgressiveId].Visibility	:= IN_Visibility;
			HMI_Data.AnalogOut[VAR_ProgressiveId].Enable		:= NOT IN_ReadOnly AND NOT IN_HMIAutoForce;
			HMI_Data.AnalogOut[VAR_ProgressiveId].PV			:= UDINT_TO_REAL(VAR_Value);
			HMI_Data.AnalogOut[VAR_ProgressiveId].Wait			:= IN_Wait;
			HMI_Data.AnalogOut[VAR_ProgressiveId].Description	:= IN_Description;
			HMI_Data.AnalogOut[VAR_ProgressiveId].Unit			:= IN_Unit;
			HMI_Data.AnalogOut[VAR_ProgressiveId].MaxValue		:= IN_MaxValue;
			HMI_Data.AnalogOut[VAR_ProgressiveId].MinValue		:= IN_MinValue;

			VAR_Man			:= HMI_Data.AnalogOut[VAR_ProgressiveId].Man;
			VAR_ManValue	:= REAL_TO_INT(HMI_Data.AnalogOut[VAR_ProgressiveId].PV_Man);
		ELSE
			HMI_Data.AnalogIn[VAR_ProgressiveId].Visibility		:= IN_Visibility;
			HMI_Data.AnalogIn[VAR_ProgressiveId].Enable			:= NOT IN_ReadOnly AND NOT IN_HMIAutoForce;
			HMI_Data.AnalogIn[VAR_ProgressiveId].PV				:= UDINT_TO_REAL(ITC);
			HMI_Data.AnalogIn[VAR_ProgressiveId].Wait			:= IN_Wait;
			HMI_Data.AnalogIn[VAR_ProgressiveId].Description	:= IN_Description;
			HMI_Data.AnalogIn[VAR_ProgressiveId].Unit			:= IN_Unit;
			HMI_Data.AnalogIn[VAR_ProgressiveId].MaxValue		:= IN_MaxValue;
			HMI_Data.AnalogIn[VAR_ProgressiveId].MinValue		:= IN_MinValue;

			VAR_Man			:= HMI_Data.AnalogIn[VAR_ProgressiveId].Man;
			VAR_ManValue	:= REAL_TO_INT(HMI_Data.AnalogIn[VAR_ProgressiveId].PV_Man);
		END_IF
	ELSIF (Index < (VAR_ProgressiveId + 4 * HMI_Page.PageNum)) THEN
		IF IN_IOType THEN
			HMI_Data.AnalogOut[VAR_ProgressiveId].Visibility	:= FALSE;
		ELSE
			HMI_Data.AnalogIn[VAR_ProgressiveId].Visibility		:= FALSE;
		END_IF
	END_IF

	VAR_OldPage := HMI_Page.PageNum;

	HMI_Data.ManActive	:= VAR_Man OR HMI_Data.ManActive;

	IF (Index > (4 + 4 * HMI_Page.PageNum)) AND IN_Visibility THEN
		HMI_Data.PageUp.Enable := TRUE;
	END_IF

	IF HMI_Page.PageNum <> 0 THEN
		HMI_Data.PageDown.Enable := TRUE;
	END_IF

	OUT_Man			:= VAR_Man;
	OUT_ManValue	:= VAR_ManValue;
	Index	:= Index + 1;
END_FUNCTION_BLOCK

FUNCTION_BLOCK FB_HMI_ITC_AnalogDIntOverUsint
	VAR_ProgressiveId := INT_TO_UINT(FC_ReminderShift(UINT_TO_INT(Index), 4, 0));

	IF IN_ReadOnly OR IN_HMIAutoForce THEN
		VAR_Man		:= FALSE;
	END_IF

	IF IN_IOType THEN
		VAR_Value		:= SEL(VAR_Man, ITC, VAR_ManValue);
		VAR_RawValue	:= SEL(HMI_Data.ComSwap, VAR_Value, swapDINT(VAR_Value));
		memcpy(ADR(ITC_IO), ADR(VAR_RawValue), SIZEOF(ITC));
	ELSE
		memcpy(ADR(VAR_RawValue), ADR(ITC_IO), SIZEOF(ITC));
		VAR_Value	:= SEL(HMI_Data.ComSwap, VAR_RawValue, swapDINT(VAR_RawValue));
		ITC			:= SEL(VAR_Man, VAR_Value, VAR_ManValue);
	END_IF

	IF VAR_OldPage <> HMI_Page.PageNum THEN
		VAR_PageSwitch	:= TRUE;
	END_IF

	IF (Index = (VAR_ProgressiveId + 4 * HMI_Page.PageNum)) AND IN_Visibility THEN
		IF VAR_PageSwitch THEN
			IF IN_IOType THEN
				HMI_Data.AnalogOut[VAR_ProgressiveId].Man		:= VAR_Man;
				HMI_Data.AnalogOut[VAR_ProgressiveId].PV_Man	:= DINT_TO_REAL(VAR_ManValue);
			ELSE
				HMI_Data.AnalogIn[VAR_ProgressiveId].Man		:= VAR_Man;
				HMI_Data.AnalogIn[VAR_ProgressiveId].PV_Man		:= DINT_TO_REAL(VAR_ManValue);
			END_IF
			VAR_PageSwitch	:= FALSE;
		END_IF

		IF IN_IOType THEN
			HMI_Data.AnalogOut[VAR_ProgressiveId].Visibility	:= IN_Visibility;
			HMI_Data.AnalogOut[VAR_ProgressiveId].Enable		:= NOT IN_ReadOnly AND NOT IN_HMIAutoForce;
			HMI_Data.AnalogOut[VAR_ProgressiveId].PV			:= DINT_TO_REAL(VAR_Value);
			HMI_Data.AnalogOut[VAR_ProgressiveId].Wait			:= IN_Wait;
			HMI_Data.AnalogOut[VAR_ProgressiveId].Description	:= IN_Description;
			HMI_Data.AnalogOut[VAR_ProgressiveId].Unit			:= IN_Unit;
			HMI_Data.AnalogOut[VAR_ProgressiveId].MaxValue		:= IN_MaxValue;
			HMI_Data.AnalogOut[VAR_ProgressiveId].MinValue		:= IN_MinValue;

			VAR_Man			:= HMI_Data.AnalogOut[VAR_ProgressiveId].Man;
			VAR_ManValue	:= REAL_TO_INT(HMI_Data.AnalogOut[VAR_ProgressiveId].PV_Man);
		ELSE
			HMI_Data.AnalogIn[VAR_ProgressiveId].Visibility		:= IN_Visibility;
			HMI_Data.AnalogIn[VAR_ProgressiveId].Enable			:= NOT IN_ReadOnly AND NOT IN_HMIAutoForce;
			HMI_Data.AnalogIn[VAR_ProgressiveId].PV				:= DINT_TO_REAL(ITC);
			HMI_Data.AnalogIn[VAR_ProgressiveId].Wait			:= IN_Wait;
			HMI_Data.AnalogIn[VAR_ProgressiveId].Description	:= IN_Description;
			HMI_Data.AnalogIn[VAR_ProgressiveId].Unit			:= IN_Unit;
			HMI_Data.AnalogIn[VAR_ProgressiveId].MaxValue		:= IN_MaxValue;
			HMI_Data.AnalogIn[VAR_ProgressiveId].MinValue		:= IN_MinValue;

			VAR_Man			:= HMI_Data.AnalogIn[VAR_ProgressiveId].Man;
			VAR_ManValue	:= REAL_TO_INT(HMI_Data.AnalogIn[VAR_ProgressiveId].PV_Man);
		END_IF
	ELSIF (Index < (VAR_ProgressiveId + 4 * HMI_Page.PageNum)) THEN
		IF IN_IOType THEN
			HMI_Data.AnalogOut[VAR_ProgressiveId].Visibility	:= FALSE;
		ELSE
			HMI_Data.AnalogIn[VAR_ProgressiveId].Visibility		:= FALSE;
		END_IF
	END_IF

	VAR_OldPage := HMI_Page.PageNum;

	HMI_Data.ManActive	:= VAR_Man OR HMI_Data.ManActive;

	IF (Index > (4 + 4 * HMI_Page.PageNum)) AND IN_Visibility THEN
		HMI_Data.PageUp.Enable := TRUE;
	END_IF

	IF HMI_Page.PageNum <> 0 THEN
		HMI_Data.PageDown.Enable := TRUE;
	END_IF

	OUT_Man			:= VAR_Man;
	OUT_ManValue	:= VAR_ManValue;
	Index			:= Index + 1;
END_FUNCTION_BLOCK

FUNCTION_BLOCK FB_HMI_ITC_AnalogReal
	VAR_ProgressiveId := INT_TO_UINT(FC_ReminderShift(UINT_TO_INT(Index), 4, 0));

	IF IN_ReadOnly OR IN_HMIAutoForce THEN
		VAR_Man		:= FALSE;
	END_IF

	IF IN_IOType THEN
		VAR_Value	:= SEL(VAR_Man, ITC, VAR_ManValue);
		ITC_IO		:= SEL(HMI_Data.ComSwap, VAR_Value, swapREAL(VAR_Value));
	ELSE
		VAR_Value	:= SEL(HMI_Data.ComSwap, ITC_IO, swapREAL(ITC_IO));
		ITC			:= SEL(VAR_Man, VAR_Value, VAR_ManValue);
	END_IF

	IF VAR_OldPage <> HMI_Page.PageNum THEN
		VAR_PageSwitch	:= TRUE;
	END_IF

	IF (Index = (VAR_ProgressiveId + 4 * HMI_Page.PageNum)) AND IN_Visibility THEN
		IF VAR_PageSwitch THEN
			IF IN_IOType THEN
				HMI_Data.AnalogOut[VAR_ProgressiveId].Man		:= VAR_Man;
				HMI_Data.AnalogOut[VAR_ProgressiveId].PV_Man	:= VAR_ManValue;
			ELSE
				HMI_Data.AnalogIn[VAR_ProgressiveId].Man	:= VAR_Man;
				HMI_Data.AnalogIn[VAR_ProgressiveId].PV_Man	:= VAR_ManValue;
			END_IF
			VAR_PageSwitch	:= FALSE;
		END_IF

		IF IN_IOType THEN
			HMI_Data.AnalogOut[VAR_ProgressiveId].Visibility	:= IN_Visibility;
			HMI_Data.AnalogOut[VAR_ProgressiveId].Enable		:= NOT IN_ReadOnly AND NOT IN_HMIAutoForce;
			HMI_Data.AnalogOut[VAR_ProgressiveId].PV			:= VAR_Value;
			HMI_Data.AnalogOut[VAR_ProgressiveId].Wait			:= IN_Wait;
			HMI_Data.AnalogOut[VAR_ProgressiveId].Description	:= IN_Description;
			HMI_Data.AnalogOut[VAR_ProgressiveId].Unit			:= IN_Unit;
			HMI_Data.AnalogOut[VAR_ProgressiveId].MaxValue		:= IN_MaxValue;
			HMI_Data.AnalogOut[VAR_ProgressiveId].MinValue		:= IN_MinValue;

			VAR_Man			:= HMI_Data.AnalogOut[VAR_ProgressiveId].Man;
			VAR_ManValue	:= HMI_Data.AnalogOut[VAR_ProgressiveId].PV_Man;
		ELSE
			HMI_Data.AnalogIn[VAR_ProgressiveId].Visibility		:= IN_Visibility;
			HMI_Data.AnalogIn[VAR_ProgressiveId].Enable			:= NOT IN_ReadOnly AND NOT IN_HMIAutoForce;
			HMI_Data.AnalogIn[VAR_ProgressiveId].PV				:= ITC;
			HMI_Data.AnalogIn[VAR_ProgressiveId].Wait			:= IN_Wait;
			HMI_Data.AnalogIn[VAR_ProgressiveId].Description	:= IN_Description;
			HMI_Data.AnalogIn[VAR_ProgressiveId].Unit			:= IN_Unit;
			HMI_Data.AnalogIn[VAR_ProgressiveId].MaxValue		:= IN_MaxValue;
			HMI_Data.AnalogIn[VAR_ProgressiveId].MinValue		:= IN_MinValue;

			VAR_Man			:= HMI_Data.AnalogIn[VAR_ProgressiveId].Man;
			VAR_ManValue	:= HMI_Data.AnalogIn[VAR_ProgressiveId].PV_Man;
		END_IF
	ELSIF (Index < (VAR_ProgressiveId + 4 * HMI_Page.PageNum)) THEN
		IF IN_IOType THEN
			HMI_Data.AnalogOut[VAR_ProgressiveId].Visibility	:= FALSE;
		ELSE
			HMI_Data.AnalogIn[VAR_ProgressiveId].Visibility		:= FALSE;
		END_IF
	END_IF

	VAR_OldPage := HMI_Page.PageNum;

	HMI_Data.ManActive	:= VAR_Man OR HMI_Data.ManActive;

	IF (Index > (4 + 4 * HMI_Page.PageNum)) AND IN_Visibility THEN
		HMI_Data.PageUp.Enable := TRUE;
	END_IF

	IF HMI_Page.PageNum <> 0 THEN
		HMI_Data.PageDown.Enable := TRUE;
	END_IF

	OUT_Man			:= VAR_Man;
	OUT_ManValue	:= VAR_ManValue;
	Index			:= Index + 1;
END_FUNCTION_BLOCK

FUNCTION_BLOCK FB_HMI_ITC_AnalogRealOverUsint
	VAR_ProgressiveId := INT_TO_UINT(FC_ReminderShift(UINT_TO_INT(Index), 4, 0));

	IF IN_ReadOnly OR IN_HMIAutoForce THEN
		VAR_Man		:= FALSE;
	END_IF

	IF IN_IOType THEN
		VAR_Value	:= SEL(VAR_Man, ITC, VAR_ManValue);
		VAR_RawValue	:= SEL(HMI_Data.ComSwap, VAR_Value, swapREAL(VAR_Value));
		memcpy(ADR(ITC_IO), ADR(VAR_RawValue), SIZEOF(ITC));
	ELSE
		memcpy(ADR(VAR_RawValue), ADR(ITC_IO), SIZEOF(ITC));
		VAR_Value	:= SEL(HMI_Data.ComSwap, VAR_RawValue, swapREAL(VAR_RawValue));
		ITC		:= SEL(VAR_Man, VAR_Value, VAR_ManValue);
	END_IF

	IF VAR_OldPage <> HMI_Page.PageNum THEN
		VAR_PageSwitch	:= TRUE;
	END_IF

	IF (Index = (VAR_ProgressiveId + 4 * HMI_Page.PageNum)) AND IN_Visibility THEN
		IF VAR_PageSwitch THEN
			IF IN_IOType THEN
				HMI_Data.AnalogOut[VAR_ProgressiveId].Man		:= VAR_Man;
				HMI_Data.AnalogOut[VAR_ProgressiveId].PV_Man	:= VAR_ManValue;
			ELSE
				HMI_Data.AnalogIn[VAR_ProgressiveId].Man		:= VAR_Man;
				HMI_Data.AnalogIn[VAR_ProgressiveId].PV_Man		:= VAR_ManValue;
			END_IF
			VAR_PageSwitch	:= FALSE;
		END_IF

		IF IN_IOType THEN
			HMI_Data.AnalogOut[VAR_ProgressiveId].Visibility	:= IN_Visibility;
			HMI_Data.AnalogOut[VAR_ProgressiveId].Enable		:= NOT IN_ReadOnly AND NOT IN_HMIAutoForce;
			VAR_Value	:= swapREAL(ITC_IO);
			memcpy(ADR(RealValue), ADR(VAR_Value), SIZEOF(RealValue));
			HMI_Data.AnalogOut[VAR_ProgressiveId].PV			:= VAR_Value;
			HMI_Data.AnalogOut[VAR_ProgressiveId].Wait			:= IN_Wait;
			HMI_Data.AnalogOut[VAR_ProgressiveId].Description	:= IN_Description;
			HMI_Data.AnalogOut[VAR_ProgressiveId].Unit			:= IN_Unit;
			HMI_Data.AnalogOut[VAR_ProgressiveId].MaxValue		:= IN_MaxValue;
			HMI_Data.AnalogOut[VAR_ProgressiveId].MinValue		:= IN_MinValue;

			VAR_Man			:= HMI_Data.AnalogOut[VAR_ProgressiveId].Man;
			VAR_ManValue	:= HMI_Data.AnalogOut[VAR_ProgressiveId].PV_Man;
		ELSE
			HMI_Data.AnalogIn[VAR_ProgressiveId].Visibility		:= IN_Visibility;
			HMI_Data.AnalogIn[VAR_ProgressiveId].Enable			:= NOT IN_ReadOnly AND NOT IN_HMIAutoForce;
			HMI_Data.AnalogIn[VAR_ProgressiveId].PV				:= ITC;
			HMI_Data.AnalogIn[VAR_ProgressiveId].Wait			:= IN_Wait;
			HMI_Data.AnalogIn[VAR_ProgressiveId].Description	:= IN_Description;
			HMI_Data.AnalogIn[VAR_ProgressiveId].Unit			:= IN_Unit;
			HMI_Data.AnalogIn[VAR_ProgressiveId].MaxValue		:= IN_MaxValue;
			HMI_Data.AnalogIn[VAR_ProgressiveId].MinValue		:= IN_MinValue;

			VAR_Man			:= HMI_Data.AnalogIn[VAR_ProgressiveId].Man;
			VAR_ManValue	:= HMI_Data.AnalogIn[VAR_ProgressiveId].PV_Man;
		END_IF
	ELSIF (Index < (VAR_ProgressiveId + 4 * HMI_Page.PageNum)) THEN
		IF IN_IOType THEN
			HMI_Data.AnalogOut[VAR_ProgressiveId].Visibility	:= FALSE;
		ELSE
			HMI_Data.AnalogIn[VAR_ProgressiveId].Visibility		:= FALSE;
		END_IF
	END_IF

	VAR_OldPage := HMI_Page.PageNum;

	HMI_Data.ManActive	:= VAR_Man OR HMI_Data.ManActive;

	IF (Index > (4 + 4 * HMI_Page.PageNum)) AND IN_Visibility THEN
		HMI_Data.PageUp.Enable := TRUE;
	END_IF

	IF HMI_Page.PageNum <> 0 THEN
		HMI_Data.PageDown.Enable := TRUE;
	END_IF

	OUT_Man			:= VAR_Man;
	OUT_ManValue	:= VAR_ManValue;
	Index			:= Index + 1;
END_FUNCTION_BLOCK

FUNCTION_BLOCK FB_HMI_ITC_End
	IF IN_IODigAnalog THEN
		VAR_ProgressiveId := INT_TO_UINT(FC_ReminderShift(UINT_TO_INT(Index), 4, 0));
		IF Index < (4 + 4 * HMI_Page.PageNum) THEN
			FOR i := Index TO (4 + Index - VAR_ProgressiveId) DO
				IF IN_IOType THEN
					HMI_Data.AnalogOut[VAR_ProgressiveId + i - Index].Visibility	:= FALSE;
				ELSE
					HMI_Data.AnalogIn[VAR_ProgressiveId + i - Index].Visibility		:= FALSE;
				END_IF
			END_FOR
		END_IF
	ELSE
		VAR_ProgressiveId := INT_TO_UINT(FC_ReminderShift(UINT_TO_INT(Index), 16, 0));
		IF Index < (16 + 16 * HMI_Page.PageNum) THEN
			FOR i := Index TO (16 + Index - VAR_ProgressiveId) DO
				IF IN_IOType THEN
					HMI_Data.DigitalOut[VAR_ProgressiveId + i - Index].Visibility	:= FALSE;
				ELSE
					HMI_Data.DigitalIn[VAR_ProgressiveId + i - Index].Visibility	:= FALSE;
				END_IF
			END_FOR
		END_IF
	END_IF
END_FUNCTION_BLOCK

FUNCTION_BLOCK FB_HMI_ITC_Start
	FOR i := 1 TO 16 DO
		HMI_Data.DigitalIn[i].Visibility	:= FALSE;
		HMI_Data.DigitalOut[i].Visibility	:= FALSE;
		IF i <= 4 THEN
			HMI_Data.AnalogOut[i].Visibility	:= FALSE;
			HMI_Data.AnalogIn[i].Visibility		:= FALSE;
		END_IF
	END_FOR

	HMI_Data.PageDown.Enable	:= FALSE;
	HMI_Data.PageUp.Enable		:= FALSE;
	HMI_Data.ManActive			:= FALSE;

	DigitalIndexIn	:= 1;
	AnalogIndexIn	:= 1;
	DigitalIndexOut	:= 1;
	AnalogIndexOut	:= 1;
END_FUNCTION_BLOCK

(* ---- FB_ITCFast.st ---- *)
FUNCTION_BLOCK FB_HMI_ITC_FastDigitalByte
	VAR_ProgressiveId := INT_TO_UINT(FC_ReminderShift(UINT_TO_INT(Index), 16, 0));

	IF IN_ReadOnly OR IN_HMIAutoForce THEN
		VAR_Auto	:= TRUE;
		VAR_Man		:= FALSE;
	END_IF

	IF VAR_OldPage <> HMI_Page.PageNum THEN
		VAR_PageSwitch	:= TRUE;
	END_IF

	IF (Index = (VAR_ProgressiveId + 16 * VAR_OldPage)) AND IN_Visibility THEN
		IF VAR_PageSwitch THEN
			IF IN_IOType THEN
				HMI_Data.DigitalOut[VAR_ProgressiveId].Auto	:= VAR_Auto;
				HMI_Data.DigitalOut[VAR_ProgressiveId].Man	:= VAR_Man;
			ELSE
				HMI_Data.DigitalIn[VAR_ProgressiveId].Auto	:= VAR_Auto;
				HMI_Data.DigitalIn[VAR_ProgressiveId].Man	:= VAR_Man;
			END_IF
			VAR_PageSwitch	:= FALSE;
		END_IF

		IF IN_IOType THEN
			HMI_Data.DigitalOut[VAR_ProgressiveId].Visibility	:= IN_Visibility;
			HMI_Data.DigitalOut[VAR_ProgressiveId].Enable		:= NOT IN_ReadOnly AND NOT IN_HMIAutoForce;
			HMI_Data.DigitalOut[VAR_ProgressiveId].LampState	:= SEL(VAR_Auto, VAR_Man, ITC);
			HMI_Data.DigitalOut[VAR_ProgressiveId].Wait			:= IN_Wait;
			HMI_Data.DigitalOut[VAR_ProgressiveId].Alarm		:= IN_Alarm;
			HMI_Data.DigitalOut[VAR_ProgressiveId].Description	:= IN_Description;

			IF EDGEPOS(HMI_Data.DigitalOut[VAR_ProgressiveId].Auto) THEN
				HMI_Data.DigitalOut[VAR_ProgressiveId].Man := FALSE;
			ELSIF EDGEPOS(HMI_Data.DigitalOut[VAR_ProgressiveId].Man) THEN
				HMI_Data.DigitalOut[VAR_ProgressiveId].Auto := FALSE;
			END_IF

			IF IN_ReadOnly OR IN_HMIAutoForce THEN
				HMI_Data.DigitalOut[VAR_ProgressiveId].Auto	:= TRUE;
				HMI_Data.DigitalOut[VAR_ProgressiveId].Man	:= FALSE;
			END_IF

			VAR_Auto	:= HMI_Data.DigitalOut[VAR_ProgressiveId].Auto;
			VAR_Man		:= HMI_Data.DigitalOut[VAR_ProgressiveId].Man;
		ELSE
			HMI_Data.DigitalIn[VAR_ProgressiveId].Visibility	:= IN_Visibility;
			HMI_Data.DigitalIn[VAR_ProgressiveId].Enable		:= NOT IN_ReadOnly AND NOT IN_HMIAutoForce;
			HMI_Data.DigitalIn[VAR_ProgressiveId].LampState 	:= SEL(VAR_Auto, VAR_Man, ITC);
			HMI_Data.DigitalIn[VAR_ProgressiveId].Wait			:= IN_Wait;
			HMI_Data.DigitalIn[VAR_ProgressiveId].Alarm			:= IN_Alarm;
			HMI_Data.DigitalIn[VAR_ProgressiveId].Description	:= IN_Description;

			IF EDGEPOS(HMI_Data.DigitalIn[VAR_ProgressiveId].Auto) THEN
				HMI_Data.DigitalIn[VAR_ProgressiveId].Man := FALSE;
			ELSIF EDGEPOS(HMI_Data.DigitalIn[VAR_ProgressiveId].Man) THEN
				HMI_Data.DigitalIn[VAR_ProgressiveId].Auto := FALSE;
			END_IF

			IF IN_ReadOnly OR IN_HMIAutoForce THEN
				HMI_Data.DigitalIn[VAR_ProgressiveId].Auto	:= TRUE;
				HMI_Data.DigitalIn[VAR_ProgressiveId].Man	:= FALSE;
			END_IF

			VAR_Auto	:= HMI_Data.DigitalIn[VAR_ProgressiveId].Auto;
			VAR_Man		:= HMI_Data.DigitalIn[VAR_ProgressiveId].Man;
		END_IF
	ELSIF (Index < (VAR_ProgressiveId + 16 * HMI_Page.PageNum)) THEN
		IF IN_IOType THEN
			HMI_Data.DigitalOut[VAR_ProgressiveId].Visibility	:= FALSE;
		ELSE
			HMI_Data.DigitalIn[VAR_ProgressiveId].Visibility	:= FALSE;
		END_IF
	END_IF

	VAR_OldPage := HMI_Page.PageNum;

	HMI_Data.ManActive	:= NOT VAR_Auto OR HMI_Data.ManActive;

	IF (Index > (16 + 16 * HMI_Page.PageNum)) AND IN_Visibility THEN
		HMI_Data.PageUp.Enable := TRUE;
	END_IF

	IF HMI_Page.PageNum <> 0 THEN
		HMI_Data.PageDown.Enable := TRUE;
	END_IF

	OUT_Man			:= NOT VAR_Auto;
	OUT_ManValue	:= VAR_Man;
	Index	:= Index + 1;
END_FUNCTION_BLOCK

FUNCTION_BLOCK FB_HMI_ITC_FastAnalogInt
	VAR_ProgressiveId := INT_TO_UINT(FC_ReminderShift(UINT_TO_INT(Index), 4, 0));

	IF IN_ReadOnly OR IN_HMIAutoForce THEN
		VAR_Man		:= FALSE;
	END_IF

	IF VAR_OldPage <> HMI_Page.PageNum THEN
		VAR_PageSwitch	:= TRUE;
	END_IF

	IF (Index = (VAR_ProgressiveId + 4 * VAR_OldPage)) AND IN_Visibility THEN
		IF VAR_PageSwitch THEN
			IF IN_IOType THEN
				HMI_Data.AnalogOut[VAR_ProgressiveId].Man		:= VAR_Man;
				HMI_Data.AnalogOut[VAR_ProgressiveId].PV_Man	:= INT_TO_REAL(VAR_ManValue);
			ELSE
				HMI_Data.AnalogIn[VAR_ProgressiveId].Man	:= VAR_Man;
				HMI_Data.AnalogIn[VAR_ProgressiveId].PV_Man	:= INT_TO_REAL(VAR_ManValue);
			END_IF
			VAR_PageSwitch	:= FALSE;
		END_IF

		IF IN_IOType THEN
			HMI_Data.AnalogOut[VAR_ProgressiveId].Visibility	:= IN_Visibility;
			HMI_Data.AnalogOut[VAR_ProgressiveId].Enable		:= NOT IN_ReadOnly AND NOT IN_HMIAutoForce;
			HMI_Data.AnalogOut[VAR_ProgressiveId].PV			:= SEL(VAR_Man, INT_TO_REAL(ITC), INT_TO_REAL(VAR_ManValue));
			HMI_Data.AnalogOut[VAR_ProgressiveId].Wait			:= IN_Wait;
			HMI_Data.AnalogOut[VAR_ProgressiveId].Description	:= IN_Description;
			HMI_Data.AnalogOut[VAR_ProgressiveId].Unit			:= IN_Unit;
			HMI_Data.AnalogOut[VAR_ProgressiveId].MaxValue		:= IN_MaxValue;
			HMI_Data.AnalogOut[VAR_ProgressiveId].MinValue		:= IN_MinValue;

			VAR_Man			:= HMI_Data.AnalogOut[VAR_ProgressiveId].Man;
			VAR_ManValue	:= REAL_TO_INT(HMI_Data.AnalogOut[VAR_ProgressiveId].PV_Man);
		ELSE
			HMI_Data.AnalogIn[VAR_ProgressiveId].Visibility		:= IN_Visibility;
			HMI_Data.AnalogIn[VAR_ProgressiveId].Enable			:= NOT IN_ReadOnly AND NOT IN_HMIAutoForce;
			HMI_Data.AnalogIn[VAR_ProgressiveId].PV				:= SEL(VAR_Man, INT_TO_REAL(ITC), INT_TO_REAL(VAR_ManValue));
			HMI_Data.AnalogIn[VAR_ProgressiveId].Wait			:= IN_Wait;
			HMI_Data.AnalogIn[VAR_ProgressiveId].Description	:= IN_Description;
			HMI_Data.AnalogIn[VAR_ProgressiveId].Unit			:= IN_Unit;
			HMI_Data.AnalogIn[VAR_ProgressiveId].MaxValue		:= IN_MaxValue;
			HMI_Data.AnalogIn[VAR_ProgressiveId].MinValue		:= IN_MinValue;

			VAR_Man			:= HMI_Data.AnalogIn[VAR_ProgressiveId].Man;
			VAR_ManValue	:= REAL_TO_INT(HMI_Data.AnalogIn[VAR_ProgressiveId].PV_Man);
		END_IF
	ELSIF (Index < (VAR_ProgressiveId + 4 * HMI_Page.PageNum)) THEN
		IF IN_IOType THEN
			HMI_Data.AnalogOut[VAR_ProgressiveId].Visibility	:= FALSE;
		ELSE
			HMI_Data.AnalogIn[VAR_ProgressiveId].Visibility	:= FALSE;
		END_IF
	END_IF

	VAR_OldPage := HMI_Page.PageNum;

	HMI_Data.ManActive	:= VAR_Man OR HMI_Data.ManActive;

	IF (Index > (4 + 4 * HMI_Page.PageNum)) AND IN_Visibility THEN
		HMI_Data.PageUp.Enable := TRUE;
	END_IF

	IF HMI_Page.PageNum <> 0 THEN
		HMI_Data.PageDown.Enable := TRUE;
	END_IF

	OUT_Man			:= VAR_Man;
	OUT_ManValue	:= VAR_ManValue;
	Index	:= Index + 1;
END_FUNCTION_BLOCK

FUNCTION_BLOCK FB_HMI_ITC_FastAnalogDInt
	VAR_ProgressiveId := INT_TO_UINT(FC_ReminderShift(UINT_TO_INT(Index), 4, 0));

	IF IN_ReadOnly OR IN_HMIAutoForce THEN
		VAR_Man		:= FALSE;
	END_IF

	IF VAR_OldPage <> HMI_Page.PageNum THEN
		VAR_PageSwitch	:= TRUE;
	END_IF

	IF (Index = (VAR_ProgressiveId + 4 * VAR_OldPage)) AND IN_Visibility THEN
		IF VAR_PageSwitch THEN
			IF IN_IOType THEN
				HMI_Data.AnalogOut[VAR_ProgressiveId].Man		:= VAR_Man;
				HMI_Data.AnalogOut[VAR_ProgressiveId].PV_Man	:= DINT_TO_REAL(VAR_ManValue);
			ELSE
				HMI_Data.AnalogIn[VAR_ProgressiveId].Man	:= VAR_Man;
				HMI_Data.AnalogIn[VAR_ProgressiveId].PV_Man	:= DINT_TO_REAL(VAR_ManValue);
			END_IF
			VAR_PageSwitch	:= FALSE;
		END_IF

		IF IN_IOType THEN
			HMI_Data.AnalogOut[VAR_ProgressiveId].Visibility	:= IN_Visibility;
			HMI_Data.AnalogOut[VAR_ProgressiveId].Enable		:= NOT IN_ReadOnly AND NOT IN_HMIAutoForce;
			HMI_Data.AnalogOut[VAR_ProgressiveId].PV			:= SEL(VAR_Man, DINT_TO_REAL(ITC), DINT_TO_REAL(VAR_ManValue));
			HMI_Data.AnalogOut[VAR_ProgressiveId].Wait			:= IN_Wait;
			HMI_Data.AnalogOut[VAR_ProgressiveId].Description	:= IN_Description;
			HMI_Data.AnalogOut[VAR_ProgressiveId].Unit			:= IN_Unit;
			HMI_Data.AnalogOut[VAR_ProgressiveId].MaxValue		:= IN_MaxValue;
			HMI_Data.AnalogOut[VAR_ProgressiveId].MinValue		:= IN_MinValue;

			VAR_Man			:= HMI_Data.AnalogOut[VAR_ProgressiveId].Man;
			VAR_ManValue	:= REAL_TO_INT(HMI_Data.AnalogOut[VAR_ProgressiveId].PV_Man);
		ELSE
			HMI_Data.AnalogIn[VAR_ProgressiveId].Visibility		:= IN_Visibility;
			HMI_Data.AnalogIn[VAR_ProgressiveId].Enable			:= NOT IN_ReadOnly AND NOT IN_HMIAutoForce;
			HMI_Data.AnalogIn[VAR_ProgressiveId].PV				:= SEL(VAR_Man, DINT_TO_REAL(ITC), DINT_TO_REAL(VAR_ManValue));
			HMI_Data.AnalogIn[VAR_ProgressiveId].Wait			:= IN_Wait;
			HMI_Data.AnalogIn[VAR_ProgressiveId].Description	:= IN_Description;
			HMI_Data.AnalogIn[VAR_ProgressiveId].Unit			:= IN_Unit;
			HMI_Data.AnalogIn[VAR_ProgressiveId].MaxValue		:= IN_MaxValue;
			HMI_Data.AnalogIn[VAR_ProgressiveId].MinValue		:= IN_MinValue;

			VAR_Man			:= HMI_Data.AnalogIn[VAR_ProgressiveId].Man;
			VAR_ManValue	:= REAL_TO_INT(HMI_Data.AnalogIn[VAR_ProgressiveId].PV_Man);
		END_IF
	ELSIF (Index < (VAR_ProgressiveId + 4 * HMI_Page.PageNum)) THEN
		IF IN_IOType THEN
			HMI_Data.AnalogOut[VAR_ProgressiveId].Visibility	:= FALSE;
		ELSE
			HMI_Data.AnalogIn[VAR_ProgressiveId].Visibility	:= FALSE;
		END_IF
	END_IF

	VAR_OldPage := HMI_Page.PageNum;

	HMI_Data.ManActive	:= VAR_Man OR HMI_Data.ManActive;

	IF (Index > (4 + 4 * HMI_Page.PageNum)) AND IN_Visibility THEN
		HMI_Data.PageUp.Enable := TRUE;
	END_IF

	IF HMI_Page.PageNum <> 0 THEN
		HMI_Data.PageDown.Enable := TRUE;
	END_IF

	OUT_Man			:= VAR_Man;
	OUT_ManValue	:= VAR_ManValue;
	Index	:= Index + 1;
END_FUNCTION_BLOCK

(* ---- LevelVariation.st ---- *)
(********************************************************************
 * COPYRIGHT -- Sidel S.p.A.
 ********************************************************************
 * Program: PC
 * File: Balayage_Flow_Contr.st
 * Author: Marco.Nicoli
 * Created: December 10, 2012
 ********************************************************************
 * Implementation of program PC
 ********************************************************************)

(*  *)
FUNCTION_BLOCK LevelVariation
	VAR_RTInfo(enable:=TRUE);
	VAR_Cycle:=	UDINT_TO_REAL(VAR_RTInfo.cycle_time)/1000000; //TASK CYCLE TIME EXPRESS IN µsec . VAR_Cycle IS CONVERTED IN s

	IF IN_Enable THEN
		IF Timer > IN_ControlTime THEN
			DeltaVolume := (IN_TankVolumePV - OldVolume);						//LEVEL VARIATION CONTROL
			IF DeltaVolume < -1.0 THEN
				AbsoluteError := AbsoluteError + ABS (DeltaVolume);				//WHEN VARIATION IS NEGATIVE THE ERROR INCREASE
				RestoreTime	  := 0.0;											//WHEN VARIATION IS NEGATIVE RESTORE TIME IS RESET
				RestoreError  := 0.0;											//WHEN VARIATION IS NEGATIVE RESTORE ERROR IS RESET
			ELSIF OUT_High THEN
				RestoreTime	:= LIMIT (0.0,RestoreTime + 1.0,RestoreTimeLimit);	//WHEN VARIATION IS POSITIVE RESTORE TIME INCREASE
				RestoreError:= 0.0;												//WHEN VARIATION IS NEGATIVE RESTORE ERROR IS RESET
			ELSE
				RestoreError := LIMIT (0.0,RestoreError + 1.0,RestoreErrorLimit); //WHEN NO ACTION BEFORE INCREASE ERROR
			END_IF

			IF RestoreTime >= RestoreTimeLimit THEN								//WHEN RESTORE TIME LIMIT REACHED VARIATION IS STEADY
				AbsoluteError	:= 0.0;											//RestoreTimeLimit = 50.0 -> Timer x 50 -> 200ms x 50 = 10s
				RestoreTime 	:= 0.0;
			END_IF

			IF RestoreError >= RestoreErrorLimit THEN 							//WHEN RESTORE ERROR IS REACHED ERROR IS RESET
				AbsoluteError   := 0.0;               							//RestoreErrorLimit = 50.0 -> Timer x 50 -> 200ms x 50 = 10s
				RestoreError    := 0.0;
			END_IF

			OldVolume	:= IN_TankVolumePV;										//ACTUAL VOLUME UPDATE
			Timer		:= 0.0;													//CYCLE TIME RESTART
		ELSE
			Timer := Timer + VAR_Cycle ;										//CYCLE TIME UPDATE
		END_IF
	ELSE
		Timer 			:= 0.0;
		AbsoluteError 	:= 0.0;
		RestoreTime 	:= 0.0;
		RestoreError    := 0.0;
		OldVolume 		:= IN_TankVolumePV;
	END_IF

	OUT_High	:= AbsoluteError > 3.0;											//HIGH FLOW REQUEST DUE TO PERSISTENT NEGATIVE VARIATION
	OUT_Low 	:= NOT OUT_High;												//LOW FLOW REQUEST DUE TO VARIATION IN TOLERANCE

END_FUNCTION_BLOCK
